		(*read Parametervalue*)
		3:	iReadValue	:=DWORD_TO_WORD(SHR(iParameterReadValue,((iSlaveaddress-(iParametergroup*2))-1)*16));
			IF (NOT bStart) OR ( bCycleMode) THEN
				fbParameterinterface(bStart			:=FALSE,
								stParameterBuffer	:=stParameterBuffer);
				IF (NOT fbParameterinterface.bBusy) THEN
					istate	:=10;
				END_IF
			ELSE
				istate	:=2;
			END_IF

			(*Quit*)
		10:	bBusy	:=FALSE;
			IF (NOT bStart) THEN
				istate	:=0;
			END_IF

	ELSE
		;
	END_CASE
END_FUNCTION_BLOCK

(* POU FB_ASI_Processdata_digital, ST *)
(*********************************************************************************************************

NAME..............	:	FB_Processdata_digital
DATE...............	:	21.03.2002
AUTHOR........	:	G.Sieder (Beckhoff Industrieelektronik)

DESCRIPTION:	FB for Read/Write digital data from/to one Slave

HISTORY:	
21.03.2002	gs	start coding

*********************************************************************************************************)
FUNCTION_BLOCK FB_ASI_Processdata_digital
VAR_INPUT
	iSlaveaddress		:BYTE;
	iSlavevalue			:BYTE;
	bParametermode		:BOOL;		(*0: Read, 1: Write *)
	bCycleMode			:BOOL;		(*0: Acyclic , 1:Cyclic (permanent Read/Write) *)
	bCommMode			:BOOL;		(*0: Parameterzugriff, 1: ADS*)
	bRegComm			:BOOL;		(*Registerkommunikation: 0: Parameterzugriff, 1: Registerkommunikation *)
	bmaskAccess		:BOOL;		(*0:usual access, 1:mask access*)
	bStart				:BOOL;
END_VAR
VAR_OUTPUT
	bBusy				:BOOL;
	bErr					:BOOL;
	iErrornumber			:DWORD;
	iReadValue			:BYTE;
	iParametergroup		:WORD;
END_VAR
VAR_IN_OUT
	stParameterBuffer		:ST_ParameterBuffer;
END_VAR
VAR
	fbParameterinterface	:FB_ASI_Parameterinterface;
	TrigStart				:R_TRIG;
	iParametermask		:WORD;
	bHiWord				:BOOL;
	iParametervalue		:DWORD;
	iParameterReadValue	:DWORD;
	istate				:INT;
END_VAR
	CASE istate OF

		0:	TrigStart(clk:=bStart);
			IF TrigStart.Q THEN
				bBusy		:=TRUE;
				bErr			:=FALSE;
				iErrornumber	:=0;
				istate		:=1;
			END_IF

		(*prepare Parametervalue*)
		1:	iParametervalue	:=0;
			iParametergroup	:=iSlaveaddress/8;
			(*iParametervalue	:=SHL((iParametervalue+iSlavevalue),(((iSlaveaddress-(iParametergroup*8))-1)*4));*)
			IF bmaskAccess THEN
				IF (iSlaveaddress- iParametergroup*8)> 4 THEN
					iParametermask	:=DWORD_TO_WORD(ROL(iParametervalue,16));
					bHiWord			:=TRUE;
				ELSE
					iParametermask	:=DWORD_TO_WORD(iParametervalue);
				END_IF
			END_IF
			istate	:=2;

		(*write Parametervalue*)
		2:	fbParameterinterface(iParameternumber	:=iSlaveaddress/8+16#80,
							iParametervalue		:=iParametervalue,
							stParameterBuffer		:=stParameterBuffer,
							bHiWord				:=bHiWord,
							bmaskAccess		:=bmaskAccess,
							iParametermask		:=iParametermask,
							bParametermode		:=bParametermode,
							bCycleMode			:=bCycleMode,
							bCommMode			:=bCommMode,
							bRegComm			:=bRegComm,
							bStart				:=TRUE);
			IF (NOT fbParameterinterface.bBusy) OR bCycleMode THEN
				IF fbParameterinterface.bErr THEN
					bErr			:=TRUE;
					iErrornumber	:=fbParameterinterface.iErrornumber;
					fbParameterinterface(bStart			:=FALSE,
									stParameterBuffer	:=stParameterBuffer);
					istate	:=10;
				ELSIF (NOT bParametermode) OR bCycleMode THEN
					iParameterReadValue	:=fbParameterinterface.iParameterReadvalue;
					istate	:=3;
				ELSE
					istate	:=3;
				END_IF
			END_IF

		(*read Parametervalue*)
		3:	iReadValue	:=(DWORD_TO_BYTE(SHR(iParameterReadValue,((iSlaveaddress-(iParametergroup*8))*4)))) AND 2#00001111;
			IF (NOT bStart) OR ( NOT bCycleMode) THEN
				fbParameterinterface(bStart			:=FALSE,
								stParameterBuffer	:=stParameterBuffer);
				IF (NOT fbParameterinterface.bBusy) THEN
					istate	:=10;
				END_IF
			ELSE
				istate	:=2;
			END_IF

			(*Quit*)
		10:	bBusy	:=FALSE;
			IF (NOT bStart) THEN
				istate	:=0;
			END_IF

	ELSE
		;
	END_CASE
END_FUNCTION_BLOCK

(* POU FB_ASI_Projecting, ST *)
(*********************************************************************************************************

NAME..............	:	FB_Projecting
DATE...............	:	21.03.2002
AUTHOR........	:	G.Sieder (Beckhoff Industrieelektronik)

DESCRIPTION:	FB to Read/Write Parameters for the slave-configuration 

HISTORY:	
21.03.2002	gs	start coding

*********************************************************************************************************)
FUNCTION_BLOCK FB_ASI_Projecting
VAR_INPUT
	iSlaveaddress		:BYTE;
	iParametervalue		:DWORD;
	bIOValue			:BOOL;	(*Read/Write IO-value of a slave*)
	bIDCode				:BOOL;	(*Read/Write	ID-code of a slave*)
	bReadWrite			:BOOL;	(*0: Read, 1: Write*)
	bReadLPS			:BOOL;	(*Read List of all projected Slaves*)
	bStart				:BOOL;
END_VAR
VAR_OUTPUT
	bBusy				:BOOL;
	bErr					:BOOL;
	iErrornumber			:DWORD;
	iParameterReadvalue	:BYTE;	(*IO-value or ID-code of a slave*)
	iLPS				:DWORD;
END_VAR
VAR_IN_OUT
	stParameterBuffer		:ST_ParameterBuffer;
END_VAR
VAR
	iProjectingStep	:INT;
	TrigStart			:R_TRIG;
	iAddressFactor	:BYTE;
	iParameternumber	:WORD;
	iReadValue		:DWORD;
	fbParameterinterface	:FB_ASI_Parameterinterface;
END_VAR
	CASE iProjectingStep OF

	(*Idle*)
	0:	TrigStart(clk:=bStart);
		IF TrigStart.Q THEN
			bBusy				:=TRUE;
			bErr					:=FALSE;
			iErrornumber			:=0;
			iProjectingStep		:=1;
		END_IF

	(*generate Parameternumber*)
	1:	iAddressFactor	:=iSlaveaddress / 8;
		IF bIOValue THEN
			iParameternumber	:=16#40+iAddressFactor;
		ELSIF bIDCode THEN
			iParameternumber	:=16#48+iAddressFactor;
		ELSIF bReadLPS	THEN
			iParameternumber	:=16#A8;
		END_IF
		iProjectingStep	:=2;

	(*write Parameter to ASI-Master*)
	2:	fbParameterinterface(iParameternumber	:=iParameternumber,
							iParametervalue	:=iParametervalue,
							stParameterBuffer	:=stParameterBuffer,
							bParametermode	:=bReadWrite,
							bCycleMode		:=TRUE,
							bStart			:=TRUE);
			IF (NOT fbParameterinterface.bBusy)  THEN
				IF fbParameterinterface.bErr THEN
					bErr			:=TRUE;
					iErrornumber	:=fbParameterinterface.iErrornumber;
					iProjectingStep	:=10;
				ELSE
					iReadValue	:=fbParameterinterface.iParameterReadvalue;
					iProjectingStep	:=3;
				END_IF
				fbParameterinterface(bStart			:=FALSE,
								stParameterBuffer	:=stParameterBuffer);
			END_IF

	(*generate ParameterReadvalue*)
	3:	IF bReadLPS THEN
			iParameterReadvalue	:=0;
			iLPS				:=iReadValue;
		ELSE
			iParameterReadvalue	:=DWORD_TO_BYTE(SHR(iReadValue,((iSlaveaddress-iAddressFactor*8)*4))) AND 2#00001111;
			iLPS	:=0;
		END_IF
		iProjectingStep	:=10;

	(*Quit*)
	10:	bBusy			:=FALSE;
		bStart			:=FALSE;
		iProjectingStep	:=0;

	ELSE
		;
	END_CASE
END_FUNCTION_BLOCK

(* POU FB_ASI_ReadParameter, ST *)
(*********************************************************************************************************

NAME..............	:	FB_ReadParameter
DATE...............	:	21.03.2002
AUTHOR........	:	G.Sieder (Beckhoff Industrieelektronik)

DESCRIPTION:	FB to read Parameters 

HISTORY:	
21.03.2002	gs	start coding

*********************************************************************************************************)
FUNCTION_BLOCK FB_ASI_ReadParameter
VAR_INPUT
	iParameternumber		:WORD;
	bCycleMode			:BOOL;		(*0: Acyclic , 1:Cyclic (permanent Read/Write) *)
	bStart				:BOOL;
END_VAR
VAR_OUTPUT
	bBusy				:BOOL;
	bErr					:BOOL;
	iErrornumber			:DWORD;
	iParameterReadvalue	:DWORD;
END_VAR
VAR_IN_OUT
	stParameterBuffer		:ST_ParameterBuffer;
END_VAR
VAR
	iReadStep	:INT;
	TrigStart		:R_TRIG;
	fbParameterinterface	:FB_ASI_Parameterinterface;
END_VAR
CASE iReadStep OF

	(*Idle*)
	0:	TrigStart(clk:=bStart);
		IF TrigStart.Q THEN
			bBusy				:=TRUE;
			bErr					:=FALSE;
			iErrornumber			:=0;
			iReadStep			:=1;
		END_IF

	(*wite Parameters to ASI-Master*)
	1:	fbParameterinterface(iParameternumber	:=iParameternumber,
							stParameterBuffer	:=stParameterBuffer,
							bParametermode	:=FALSE,
							bCycleMode		:=bCycleMode,
							bStart			:=TRUE);
		(*read Parameters *)
		IF (NOT fbParameterinterface.bBusy) OR  bCycleMode THEN
			IF fbParameterinterface.bErr THEN
				bErr			:=TRUE;
				iErrornumber	:=fbParameterinterface.iErrornumber;
				iReadStep	:=5;
			ELSE
				iParameterReadvalue	:=fbParameterinterface.iParameterReadvalue;
				IF (NOT bCycleMode) OR (NOT bStart) THEN
					iReadStep	:=5;
				ELSE
					iReadStep	:=1;
				END_IF
			END_IF
		END_IF

	5:	fbParameterinterface(bStart			:=FALSE,
						stParameterBuffer	:=stParameterBuffer);
		IF (NOT fbParameterinterface.bBusy) THEN
			iReadStep	:=10;
		END_IF

	(*Quit*)
	10:	bBusy			:=FALSE;
		bStart			:=FALSE;
		iReadStep	:=0;

	ELSE
		;
	END_CASE
END_FUNCTION_BLOCK

(* POU FB_ASI_SlaveDiag, ST *)
(*********************************************************************************************************

NAME..............	:	FB_WriteParameter
DATE...............	:	21.03.2002
AUTHOR........	:	G.Sieder (Beckhoff Industrieelektronik)

DESCRIPTION:	FB for cyclic slave-diagnosis

HISTORY:	
21.03.2002	gs	start coding
03.09.2002	gs	replace bStop by bCycleMode
*********************************************************************************************************)
FUNCTION_BLOCK FB_ASI_SlaveDiag
VAR_INPUT
	iSlaveaddress		:BYTE;
	iCounter				:INT;		(*1:PhysicalFaultCounter,  2:TimeoutCounter,  3:ResponseCounter,  4:Leave-DataExchCounter,  5:DataExch-FailedCounter *)
	bCounterReset		:BOOL;
	bReadLES			:BOOL;		(*Read List of all detected Slaves*)
	bReadLAS			:BOOL;		(*Read List of all activated Slaves*)
	bCycleMode			:BOOL;		(*0: Acyclic , 1:Cyclic (permanent Read/Write) *)
	bStart				:BOOL;

END_VAR
VAR_OUTPUT
	bBusy				:BOOL;
	bErr					:BOOL;
	iErrornumber			:DWORD;
	iCounterValue		:WORD;		(*Counter of a slave*)
	iSlaveList			:DWORD;	(*LES or LAS of all Slaves*)
END_VAR
VAR_IN_OUT
	stParameterBuffer		:ST_ParameterBuffer;
END_VAR
VAR
	iDiagStep			:INT;
	TrigStart				:R_TRIG;
	iAddressFactor		:BYTE;
	iParameternumber		:WORD;
	iReadValue			:DWORD;
	fbParameterinterface	:FB_ASI_Parameterinterface;

	TimerResetCounter	:TON;
END_VAR
	CASE iDiagStep OF

	(*Idle*)
	0:	TrigStart(clk:=bStart);
		IF TrigStart.Q THEN
			bBusy				:=TRUE;
			bErr					:=FALSE;
			iErrornumber			:=0;
			iDiagStep			:=1;
		END_IF

	(*generate Parameternumber*)
	1:	iAddressFactor	:=iSlaveaddress / 2;
		IF bReadLES	THEN
			iParameternumber	:=16#B0;
		ELSIF bReadLAS THEN
			iParameternumber	:=16#B8;
		ELSE
			CASE iCounter OF
				1:	iParameternumber	:=16#140+iAddressFactor;
				2:	iParameternumber	:=16#160+iAddressFactor;
				3:	iParameternumber	:=16#180+iAddressFactor;
				4:	iParameternumber	:=16#1A0+iAddressFactor;
				5:	iParameternumber	:=16#1C0+iAddressFactor;
			ELSE
				;
			END_CASE
		END_IF
		iDiagStep	:=2;

	(*write Parameter to ASI-Master*)
	2:	fbParameterinterface(iParameternumber		:=iParameternumber,
							stParameterBuffer		:=stParameterBuffer,
							iParametervalue		:=0,
							bParametermode		:=bCounterReset,
							bCycleMode			:=TRUE,
							bStart				:=TRUE);
				IF fbParameterinterface.bErr THEN
					bErr			:=TRUE;
					iErrornumber	:=fbParameterinterface.iErrornumber;
					iDiagStep	:=10;
				ELSE
					iReadValue	:=fbParameterinterface.iParameterReadvalue;
					iDiagStep	:=3;
				END_IF
				TimerResetCounter(in:=bCounterReset,pt:=t#200ms);
				IF TimerResetCounter.Q THEN
					bCounterReset		:=FALSE;
					TimerResetCounter.IN 	:=FALSE;
				END_IF

	(*generate ParameterReadvalue*)
	3:	fbParameterinterface(stParameterBuffer	:=stParameterBuffer);
		IF bReadLES OR bReadLAS THEN
			iCounterValue	:=0;
			iSlaveList		:=iReadValue;
		ELSE
			iCounterValue	:=DWORD_TO_WORD(SHR(iReadValue,((iSlaveaddress-iAddressFactor*2)*16)));
			iSlaveList	:=0;
		END_IF
		IF (NOT bStart) THEN
			fbParameterinterface(bStart	:=FALSE,
							stParameterBuffer	:=stParameterBuffer);
			IF (NOT fbParameterinterface.bBusy) THEN
				iDiagStep	:=10;
			END_IF
		ELSE
			iDiagStep	:=2;
		END_IF

	(*Quit*)
	10:	bBusy		:=FALSE;
		bStart		:=FALSE;
		iDiagStep	:=0;

	ELSE
		;
	END_CASE
END_FUNCTION_BLOCK

(* POU FB_ASI_WriteParameter, ST *)
(*********************************************************************************************************

NAME..............	:	FB_WriteParameter
DATE...............	:	21.03.2002
AUTHOR........	:	G.Sieder (Beckhoff Industrieelektronik)

DESCRIPTION:	FB to write Parameters 

HISTORY:	
21.03.2002	gs	start coding
03.09.2002	gs	Output ReadValue removed
*********************************************************************************************************)
FUNCTION_BLOCK FB_ASI_WriteParameter
VAR_INPUT
	iParameternumber		:WORD;
	iParametervalue		:DWORD;
	bStart				:BOOL;
END_VAR
VAR_OUTPUT
	bBusy				:BOOL;
	bErr					:BOOL;
	iErrornumber			:DWORD;
END_VAR
VAR_IN_OUT
	stParameterBuffer		:ST_ParameterBuffer;
END_VAR
VAR
	iWriteStep	:INT;
	TrigStart		:R_TRIG;
	fbParameterinterface	:FB_ASI_Parameterinterface;
END_VAR
	CASE iWriteStep OF

	(*Idle*)
	0:	TrigStart(clk:=bStart);
		IF TrigStart.Q THEN
			bBusy				:=TRUE;
			bErr					:=FALSE;
			iErrornumber			:=0;
			iWriteStep			:=1;
		END_IF

	(*wite Parameters to ASI-Master*)
	1:	fbParameterinterface(iParameternumber	:=iParameternumber,
							iParametervalue	:=iParametervalue,
							stParameterBuffer	:=stParameterBuffer,
							bParametermode	:=TRUE,
							bCycleMode		:= FALSE,
							bStart			:=TRUE);
		IF  fbParameterinterface.bBusy  THEN
			iWriteStep	:=5;
		END_IF


	5:	fbParameterinterface(stParameterBuffer	:=stParameterBuffer);
		IF (NOT fbParameterinterface.bBusy) THEN
			IF fbParameterinterface.bErr THEN
				bErr			:=TRUE;
				iErrornumber	:=fbParameterinterface.iErrornumber;
			END_IF
			iWriteStep	:=10;
		END_IF

	(*Quit*)
	10:	bBusy			:=FALSE;
		bStart			:=FALSE;
		iWriteStep	:=0;

	ELSE
		;
	END_CASE
END_FUNCTION_BLOCK

(* POU FB_ASI_WriteReadParameter, ST *)
(*********************************************************************************************************

NAME..............	:	FB_WriteReadParameter
DATE...............	:	18.08.2003
AUTHOR........	:	G.Sieder (Beckhoff Industrieelektronik)

DESCRIPTION:	FB to write Parameters with answer 

HISTORY:	
18.08.2003	gs	start coding

*********************************************************************************************************)
FUNCTION_BLOCK FB_ASI_WriteReadParameter
VAR_INPUT
	iParameternumber		:WORD;
	iParametervalue		:DWORD;
	bStart				:BOOL;
END_VAR
VAR_OUTPUT
	bBusy				:BOOL;
	bErr					:BOOL;
	iParameterReadValue	:DWORD;
	iErrornumber			:DWORD;
END_VAR
VAR_IN_OUT
	stParameterBuffer		:ST_ParameterBuffer;
END_VAR
VAR
	iWriteStep	:INT;
	TrigStart		:R_TRIG;
	fbParameterinterface	:FB_ASI_Parameterinterface;
END_VAR
	CASE iWriteStep OF

	(*Idle*)
	0:	TrigStart(clk:=bStart);
		IF TrigStart.Q THEN
			bBusy				:=TRUE;
			bErr					:=FALSE;
			iErrornumber			:=0;
			iWriteStep			:=1;
		END_IF

	(*wite Parameters to ASI-Master*)
	1:	fbParameterinterface(iParameternumber	:=iParameternumber,
							iParametervalue	:=iParametervalue,
							stParameterBuffer	:=stParameterBuffer,
							bParametermode	:=TRUE,
							bCycleMode		:= FALSE,
							bStart			:=TRUE);
		IF  fbParameterinterface.bBusy  THEN
			iWriteStep	:=5;
		END_IF


	5:	fbParameterinterface(stParameterBuffer	:=stParameterBuffer);
		IF (NOT fbParameterinterface.bBusy) THEN
			IF fbParameterinterface.bErr THEN
				bErr			:=TRUE;
				iErrornumber	:=fbParameterinterface.iErrornumber;
				iParameterReadValue	:=0;
			ELSE
				iParameterReadValue	:=fbParameterinterface.iParameterReadvalue;
			END_IF
			iWriteStep	:=10;
		END_IF

	(*Quit*)
	10:	bBusy			:=FALSE;
		bStart			:=FALSE;
		iWriteStep	:=0;

	ELSE
		;
	END_CASE
END_FUNCTION_BLOCK

(* POU FB_AX2000_AXACT, ST *)
FUNCTION_BLOCK FB_AX2000_AXACT
VAR_INPUT
	bMode_DigitalSpeed	: BOOL;			(*OP-Mode digital speed instead of Positioning*)
	iDigitalSpeed			: DWORD;			(*digital speed if OP-Mode = digital speed*)
	iVelocity				: DWORD;		(*Velocity*)
	iPosition				: DINT;			(*Position*)
	imotion_tasknumber	: WORD;			(*number of EEPROM-saved motion-task*)
	imotion_blocktype		: WORD;			(*optional Parameters of motion tasks*)
	bStart				: BOOL;			(*START*)
	bStop				: BOOL;			(*STOP*)
	bShortStop			: BOOL;			(*1: break of motion task, 0: continue same motion task*)
	bErrorResume		: BOOL;			(*Error resume*)
	tTimeOut				: TIME:=t#5s;
END_VAR
VAR_OUTPUT

	bBusy				: BOOL;
	bError				: BOOL;			(*Errorstatus of Servo*)
	bTimeOutErr			: BOOL;

END_VAR
VAR
	i16State:				INT;
	icheckStatus:			WORD;
	icheckControlWord:	WORD;			(*ControlWord for Servo*)

	bServoReady:		BOOL;			(*readyFlag for HSW*)
	TrigStart:				R_TRIG;
	TrigTimeOut:			R_TRIG;
	bResetServo:			BOOL;			(*first move of Servo after Start/Restart*)

	TimerTimeOut		:TON;
	bTimeOutStart		:BOOL;

	iHighByte			:BYTE;
	iLowByte				:BYTE;
	icheckByteSwaping	:WORD;
	bMapInOutputs		:BOOL;
	bShortStop_check		:BOOL;

	(*virtual Input/Output*)
	stPZD_IN:		ST_PZD_IN;
	stPZD_OUT:		ST_PZD_OUT;
END_VAR
VAR_IN_OUT
	stPZDIN:		ST_PZD_IN;			(*Data from NC*)
	stPZDOUT:		ST_PZD_OUT;			(*Data to NC*)
END_VAR
	a_MapInputs();			(*mapping of real Inputs to virtual Inputs by swaping LowByte and HighByte*)
	a_RW_CtrlWord();			(*AXACT-controls*)
	a_MapOutputs();			(*mapping of virtual Outputs to real Outputs by swaping LowByte and HighByte*)
END_FUNCTION_BLOCK
ACTION a_MapInputs:
stPZD_IN.wSTW		:=ROL(stPZDIN.wSTW,8);
stPZD_IN.wHIW		:=ROL(stPZDIN.wHIW,8);
stPZD_IN.PZD3		:=ROL(stPZDIN.PZD3,8);
stPZD_IN.PZD4		:=ROL(stPZDIN.PZD4,8);
stPZD_IN.PZD5		:=ROL(stPZDIN.PZD5,8);
stPZD_IN.PZD6		:=ROL(stPZDIN.PZD6,8);
END_ACTION
ACTION a_MapOutputs:
IF bMapInOutputs THEN
	stPZDOUT.wCtrlW		:=ROL(stPZD_OUT.wCtrlW,8);
	stPZDOUT.PZD2		:=ROL(stPZD_OUT.PZD2,8);
	stPZDOUT.PZD3		:=ROL(stPZD_OUT.PZD3,8);
	stPZDOUT.PZD4		:=ROL(stPZD_OUT.PZD4,8);
	stPZDOUT.PZD5		:=ROL(stPZD_OUT.PZD5,8);
	stPZDOUT.PZD6		:=ROL(stPZD_OUT.PZD6,8);
END_IF
END_ACTION
ACTION a_RW_CtrlWord:
	bMapInOutputs	:= TRUE;

	(* Errorstatus*)
	icheckStatus:=2#00000000_00001000;
	IF (stPZD_IN.wSTW AND icheckStatus)<>0 THEN
		i16State:=10;
	END_IF

	(*short break of a motion task*)
	IF bShortStop AND (NOT bShortStop_check)THEN
		stPZD_OUT.wCtrlW:=stPZD_OUT.wCtrlW AND 2#1111111111011111;
		bShortStop_check	:=TRUE;
	ELSIF (NOT bShortStop) AND bShortStop_check THEN
		bShortStop_check	:=FALSE;
		IF (NOT bStart) THEN
			i16State			:= 11;
			bBusy			:= FALSE;
		ELSE
			stPZD_OUT.wCtrlW:=stPZD_OUT.wCtrlW OR 2#0000000000100000;
		END_IF
	END_IF

	(*Stophandling*)
	IF  bStop THEN
		stPZD_OUT.wCtrlW:=2#0000000000000101;
		bBusy			:= FALSE;
		bStart			:= FALSE;
		bMapInOutputs	:= TRUE;
		i16State			:= 11;
	END_IF

	(*TimeOut*)
	IF (NOT bMode_DigitalSpeed) THEN
		TrigTimeOut(clk:=bStart);
		IF TrigTimeOut.Q THEN
			bTimeOutStart	:=TRUE;
			bTimeOutErr		:= FALSE;
			bError			:= FALSE;
		END_IF
		IF bBusy THEN
			TimerTimeOut(IN:= FALSE, PT:= tTimeOut );
			bTimeOutStart	:=FALSE;
		ELSE
			TimerTimeOut(IN:= bTimeOutStart, PT:= tTimeOut );
		END_IF
		IF TimerTimeOut.Q THEN
			bTimeOutErr		:=TRUE;
			bTimeOutStart	:= FALSE;
			bServoReady	:= FALSE;
			i16State			:= 11;
		END_IF
	END_IF

	CASE i16State OF

		(*Initialisierung*)
	0:	bServoReady:= 	FALSE;
		bResetServo:=	TRUE;
		i16State:= i16State+1;

		(*Einschaltsperre*)
	1:	stPZD_OUT.wCtrlW:=2#0000000000000000;
		icheckStatus:=2#0000000001000000;
		IF (stPZD_IN.wSTW AND icheckStatus)<>0 THEN
			stPZD_OUT.wCtrlW:=2#0000000000000110;
			bServoReady:= FALSE;
			i16State:= i16State+1;
		END_IF

		(*einschaltbereit*)
	2:	icheckStatus:=2#0000001000000001;
		IF (stPZD_IN.wSTW AND icheckStatus)<>0 THEN
			stPZD_OUT.wCtrlW:=2#0000000000000111;
			bServoReady:= FALSE;
			i16State:= i16State+1;
		END_IF

		(*betriebsbereit*)
	3:	icheckStatus:=2#0000001000100011;
		IF (stPZD_IN.wSTW AND icheckStatus)<>0 THEN
			stPZD_OUT.wCtrlW:=2#0000010000111111;
			i16State:= i16State+1;
		END_IF

		(*Betrieb freigegeben*)
	4:	icheckStatus:=2#0000001000100111;
		IF (stPZD_IN.wSTW AND icheckStatus)<>0 THEN
			i16State:= i16State+1;
		END_IF

		(*benutzerdefinierte Daten übertragen*)
	5:	TrigStart(clk:=bStart);
		bMapInOutputs	:= FALSE;
		IF TrigStart.Q THEN
			bMapInOutputs:= TRUE;
			a_RW_PZD();
			bError		:= FALSE;
			bTimeOutErr	:= FALSE;
			bResetServo	:= FALSE;
		END_IF
		IF (NOT bResetServo) THEN
			icheckStatus:=2#0010000000000000;
			IF (stPZD_IN.wSTW AND icheckStatus)<>0 THEN
				;
			ELSE
				bBusy	:= TRUE;
				i16State:= 6;
			END_IF
		END_IF

	6:	icheckStatus:=2#0010000000000000;
		IF (stPZD_IN.wSTW AND icheckStatus)<>0 THEN
			bBusy	:= FALSE;
			i16State:= 5;
		END_IF
		IF bMode_DigitalSpeed THEN
			stPZD_OUT.PZD3	:=DWORD_TO_WORD(iDigitalSpeed*140);
			stPZD_OUT.PZD2	:=DWORD_TO_WORD(SHR((iDigitalSpeed*140),16));
		END_IF

		(* Errorhandling*)
	10:	bError			:= TRUE;
		bBusy			:= FALSE;
		bServoReady	:= FALSE;
		IF BErrorResume THEN
			stPZD_OUT.wCtrlW:=2#0000010010001111;
			i16State:=11;
		END_IF

	11:	IF (NOT bStart) THEN
			i16State:=0;
		END_IF

END_CASE
END_ACTION
ACTION a_RW_PZD:
IF bMode_DigitalSpeed THEN
	stPZD_OUT.PZD3	:=DWORD_TO_WORD(iDigitalSpeed*140);
	stPZD_OUT.PZD2	:=DWORD_TO_WORD(SHR((iDigitalSpeed*140),16));
	icheckControlWord:=2#0000000001000000;
	IF (icheckControlWord AND stPZD_OUT.wCtrlW)<>0 THEN
		stPZD_OUT.wCtrlW:=16#443F;
	ELSE
		stPZD_OUT.wCtrlW:=16#447F;
	END_IF
ELSIF (imotion_tasknumber <> 0) THEN
	stPZD_OUT.PZD2	:=imotion_tasknumber;
	icheckControlWord:=2#0000000001000000;
	IF (icheckControlWord AND stPZD_OUT.wCtrlW)<>0 THEN
		stPZD_OUT.wCtrlW:=16#043F;
	ELSE
		stPZD_OUT.wCtrlW:=16#047F;
	END_IF
ELSIF (iVelocity<>0) THEN
	stPZD_OUT.PZD3	:=DWORD_TO_WORD(iVelocity);
	stPZD_OUT.PZD2	:=DWORD_TO_WORD(SHR(iVelocity,16));
	stPZD_OUT.PZD5	:=DWORD_TO_WORD(DINT_TO_DWORD( iPosition ));
	stPZD_OUT.PZD4	:=DWORD_TO_WORD(SHR(DINT_TO_DWORD( iPosition ),16));
	stPZD_OUT.PZD6	:=imotion_blocktype;
	icheckControlWord:=2#0000000001000000;
	IF (icheckControlWord AND stPZD_OUT.wCtrlW)<>0 THEN
		stPZD_OUT.wCtrlW:=16#443F;
	ELSE
		stPZD_OUT.wCtrlW:=16#447F;
	END_IF
END_IF
END_ACTION

(* POU FB_AX2000_JogMode, ST *)
FUNCTION_BLOCK FB_AX2000_JogMode
VAR_INPUT
	bStart		: BOOL;
	bStop		: BOOL;
	iBasicVelo	: INT;				(*BasicVelocity*)
	tTimeOut		: TIME:=t#5s;

END_VAR
VAR_OUTPUT
	bBusy		: BOOL;
	bErr			: BOOL;
	bTimeOutErr	: BOOL;

END_VAR
VAR_IN_OUT
	stPZDIN			: ST_PZD_IN;			(*Data from NC*)
	stPZDOUT		: ST_PZD_OUT;		(*Data to NC*)
END_VAR
VAR
	i16state			: INT;

	icheckStatus		: DWORD;
	TrigTimeOut		: R_TRIG;
	bTimeOutStart	: BOOL;
	TimerTimeOut	: TON;
	bMapInOutputs	: BOOL;
	(*virtual Input/Output*)
	stPZD_IN:		ST_PZD_IN;
	stPZD_OUT:		ST_PZD_OUT;

END_VAR
	a_MapInputs();

	(* Errorstatus*)
	icheckStatus:=2#00000000_00001000;
	IF (stPZD_IN.wSTW AND icheckStatus)<>0 THEN
		bErr	:= TRUE;
		i16State:=10;
	END_IF

	(*TimeOut*)
	TrigTimeOut(clk:=bStart);
	IF TrigTimeOut.Q THEN
		bTimeOutStart	:=TRUE;
	END_IF
	IF bBusy THEN
		TimerTimeOut(IN:= FALSE, PT:= tTimeOut );
		bTimeOutStart	:=FALSE;
	ELSE
		TimerTimeOut(IN:= bTimeOutStart, PT:= tTimeOut );
	END_IF
	IF TimerTimeOut.Q THEN
		TimerTimeOut(IN:= FALSE, PT:= tTimeOut );
		bTimeOutErr		:=TRUE;
		bTimeOutStart	:= FALSE;
		i16State			:= 10;
	END_IF

	CASE i16state OF

	0:	IF bStart THEN
			bErr				:= FALSE;
			bTimeOutErr		:= FALSE;
			i16state			:= 1;
		END_IF

	1:	stPZD_OUT.PZD2	:=iBasicVelo;
		stPZD_OUT.wCtrlW:=(ROL(stPZDOUT.wCtrlW,8))+16#100;
		bMapInOutputs	:= TRUE;
		i16state	:= 2;

	2:	icheckStatus:=2#00100010_00000000;
		IF (stPZD_IN.wSTW AND icheckStatus)=0 OR  (stPZD_IN.wSTW AND icheckStatus)=16#2200 THEN
			;
		ELSE
			bBusy	:=TRUE;
			i16state	:= 3;
		END_IF

	3:	IF bStop THEN
			stPZD_OUT.wCtrlW:=(ROL(stPZDOUT.wCtrlW,8))-16#100;
			i16state	:= 10;
		END_IF

	10:	bBusy			:=FALSE;
		bMapInOutputs	:=FALSE;
		IF (NOT bstart) THEN
			i16state	:= 0;
		END_IF

	END_CASE

	a_MapOutputs();
END_FUNCTION_BLOCK
ACTION a_MapInputs:
	stPZD_IN.wSTW		:=ROL(stPZDIN.wSTW,8);
	stPZD_IN.wHIW		:=ROL(stPZDIN.wHIW,8);
	stPZD_IN.PZD3		:=ROL(stPZDIN.PZD3,8);
	stPZD_IN.PZD4		:=ROL(stPZDIN.PZD4,8);
	stPZD_IN.PZD5		:=ROL(stPZDIN.PZD5,8);
	stPZD_IN.PZD6		:=ROL(stPZDIN.PZD6,8);
END_ACTION
ACTION a_MapOutputs:
IF bMapInOutputs THEN
	stPZDOUT.wCtrlW		:=ROL(stPZD_OUT.wCtrlW,8);
	stPZDOUT.PZD2		:=ROL(stPZD_OUT.PZD2,8);
	stPZDOUT.PZD3		:=ROL(stPZD_OUT.PZD3,8);
	stPZDOUT.PZD4		:=ROL(stPZD_OUT.PZD4,8);
	stPZDOUT.PZD5		:=ROL(stPZD_OUT.PZD5,8);
	stPZDOUT.PZD6		:=ROL(stPZD_OUT.PZD6,8);
END_IF
END_ACTION

(* POU FB_AX2000_Parameter, ST *)
FUNCTION_BLOCK FB_AX2000_Parameter
VAR_INPUT
	iSlaveAddress:	BYTE := 0;			(* Station Address of the Slave *)
	iPnu:				WORD := 16#03A2;	(* Parameter-Number *)
	nAxis:				BYTE := 1;			(* Number of Axis *)
	iLength:			BYTE := 4;			(* Length of the parameter (2 or 4) *)
	iSubindex:			BYTE := 1;			(*Subindex*)
	iParameterValue:	DWORD := 2;			(* Parameter value *)
	iFC310xDeviceId: 	WORD := 1;			(* Device-ID of the FCxxxx *)
	bStartRead:		BOOL;				(* StartFlag to start the PKW-Read *)
	bStartWrite:		BOOL;				(* StartFlag to start the PKW-Write *)
	tTimeOut:			TIME := DEFAULT_ADS_TIMEOUT;
END_VAR
VAR_OUTPUT
	bBusy				:BOOL;
	iErrorId			:DWORD;
	iReadValue		:DINT;
END_VAR
VAR
	iError:					DWORD;
	fbReadPkw:				FB_FCxxxxDpv0PkwRead;
	fbWritePkw: 				FB_FCxxxxDpv0PkwWrite;

END_VAR
IF bStartRead OR bStartWrite THEN
	IF iLength<>2 THEN
		iLength:= 4;
	END_IF
	
	(* PKW-Read with DPV0  for Stoever-Drive (ArrayCodesNotSupported and Subindex in Octet 3 must be set) *)
	fbReadPkw(bStartFlag := bStartRead, iStationAdd := iSlaveAddress, iDeviceId := iFC310xDeviceId,nAxis := nAxis, iPnu := iPnu, iSubindex := iSubindex, iLength := iLength, bArrayCodesNotSupported := TRUE, bSubindexInOctet3 := TRUE, tTimeOut:=tTimeOut);
	IF (bStartRead AND NOT fbReadPkw.bBusy) THEN
		iError := fbReadPkw.iErrorId;
		iReadValue := fbReadPkw.iReadValue;
		bStartRead := FALSE;
	END_IF;
	
	(* PKW-Write with DPV0  for Stoever-Drive (ArrayCodesNotSupported and Subindex in Octet 3 must be set) *)
	fbWritePkw(bStartFlag := bStartWrite, iStationAdd := iSlaveAddress, iDeviceId := iFC310xDeviceId, nAxis := nAxis, iPnu := iPnu, iSubindex := iSubindex, iLength := iLength, iWriteValue := iParameterValue, bArrayCodesNotSupported := TRUE, bSubindexInOctet3 := TRUE, tTimeOut:=tTimeOut);
	IF (bStartWrite AND NOT fbWritePkw.bBusy) THEN
		iError := fbWritePkw.iErrorId;
		bStartWrite := FALSE;
	END_IF;

	bBusy:=fbReadPkw.bBusy OR fbWritePkw.bBusy;
	iErrorId:=iError;
	(*iReadValue:=iParameterValue;*)
END_IF
END_FUNCTION_BLOCK

(* POU FB_FCxxxxDpv0PkwRead, ST *)
FUNCTION_BLOCK FB_FCxxxxDpv0PkwRead
VAR_INPUT
	bStartFlag:BOOL;					(* StartFlag to start the PKW-Read *)
	iStationAdd: BYTE;				(* Station Address of the Slave *)
	iDeviceId: WORD;					(* Device-ID of the FCxxxx *)
	nAxis: BYTE;						(* Number of Axis *)
	iPnu: WORD;						(* Parameter-Number *)
	iSubindex: BYTE;					(* Subindex  *)
	iLength:BYTE;					(* Length of the parameter (2 or 4) *)
	bArrayCodesNotSupported: BOOL;	(* if the drive does not support the ARRAY-AKs 6,7 and 8, this flag should be set (then the AKs 1,2,3 will be used for Arrays) *)
	bSubindexInOctet3:BOOL;			(* if the drive needs the subindex in Octet 3 (ProfiDrive 2.0), this flag should be set *)
	tTimeOut		: TIME;
END_VAR
VAR_OUTPUT
	bBusy:BOOL;			(* Reading is busy *)
	iErrorId:DWORD;
	iReadValue:DWORD;	(* Parameter value *)
END_VAR
VAR
	fbRead:ADSREAD;
	fbDevNetId:IOF_GetDeviceNetId;
	istate:WORD := 0;
	sDevNetId:STRING(23);
	iIdxGrp: DWORD;
	iport:WORD;
	iParameterValue:DWORD;
END_VAR
CASE istate OF

	0:	(*Idle*)
		IF bStartFlag THEN
			bBusy	:=TRUE;
			istate := 1;
		END_IF

	1:	(* Get Net-ID of FCxxxx-Device *)
		fbDevNetId(NETID := '', DEVICEID := iDeviceId, START := TRUE,  TMOUT := T#1s);
		IF (NOT fbDevNetId.BUSY) THEN
			IF (NOT fbDevNetId.Err) THEN
				sDevNetId := fbDevNetId.DeviceNetId;
				istate := 2;
			ELSE
				iErrorId		:=fbDevNetId.ERRID;
				bStartFlag	:=FALSE;
				bBusy		:=FALSE;
				istate := 0;
			END_IF
			fbDevNetId(NETID := '', DEVICEID := iDeviceId, START := FALSE,  TMOUT := T#1s);
		END_IF

	2:	(* Read Parameter if StartFlag is set *)
		iport := iStationAdd;
		iport := iport + 16#1000;
		iIdxGrp := nAxis;
		iIdxGrp := SHL(iIdxGrp, 28);
		iIdxGrp := iIdxGrp +iPnu;
		IF (bArrayCodesNotSupported) THEN
			iIdxGrp := iIdxGrp + 16#8000000;
		END_IF
		IF (bSubindexInOctet3) THEN
			iIdxGrp := iIdxGrp + 16#4000000;
		END_IF
		fbRead(	NETID := sDevNetId, PORT := iport, IDXGRP := iIdxGrp, IDXOFFS := iSubindex, LEN := iLength,
				DESTADDR := ADR(iParameterValue), READ := bStartFlag, TMOUT := tTimeOut);
		istate := 3;

	3:	fbRead(	NETID := sDevNetId, PORT := iport, IDXGRP := iIdxGrp, IDXOFFS := iSubindex, LEN := iLength,
				DESTADDR := ADR(iParameterValue), READ := bStartFlag, TMOUT := tTimeOut);
		IF (NOT FbRead.BUSY) OR fbRead.Err THEN
			iErrorId := FbRead.ERRID;
			iReadValue := iParameterValue;
			istate := 4;
		END_IF

	4:	(* There must be a rising edge on the READ-input of ADSREAD to start the next reading *)
		fbRead(	NETID := sDevNetId, PORT := iport, IDXGRP := iIdxGrp, IDXOFFS := iSubindex, LEN := iLength,
				DESTADDR := ADR(iParameterValue), READ := FALSE, TMOUT := tTimeOut);
		bBusy 		:= FALSE;
		bStartFlag	:= FALSE;
		istate := 0;
END_CASE
END_FUNCTION_BLOCK

(* POU IOF_GetDeviceNetId, ST *)
FUNCTION_BLOCK IOF_GetDeviceNetId
VAR_INPUT
	NETID		: T_AmsNetId;
	DEVICEID	: UDINT;
	START		: BOOL;
	TMOUT		: TIME := DEFAULT_ADS_TIMEOUT;
END_VAR
VAR_OUTPUT
	BUSY		: BOOL;
	ERR			: BOOL;
	ERRID		: UDINT;
	DeviceNetId	: T_AmsNetId;
END_VAR
{library private}
VAR
	ADSREADEX1	: ADSREADEX := ( PORT:= AMSPORT_R0_IO, IDXOFFS:= 16#00000005 );
	RisingEdge	: R_TRIG;
	state		: BYTE;
	tmpNetId	: ARRAY[0..5] OF BYTE;
END_VAR
RisingEdge( CLK:=START );
IF RisingEdge.Q THEN
	state := 1;
END_IF
CASE state OF
	0:;(* idle state *)
	1:
		BUSY := TRUE;
		ERR := FALSE;
		ERRID := 0;
		DeviceNetId := '';
		MEMSET( ADR( tmpNetId ), 0, SIZEOF( tmpNetId ) );
		IF ( DEVICEID > 0 ) THEN
			ADSREADEX1( READ:=FALSE );
			ADSREADEX1( NETID:=NETID, IDXGRP:= 16#00005000 + DEVICEID,
						LEN:= SIZEOF( tmpNetId ), DESTADDR:= ADR( tmpNetId ),
						READ:=TRUE, TMOUT:= TMOUT );
			state := 2;
		ELSE
			ERR := TRUE;
			ERRID :=16#706;	(* Parameter value not correct! *)
			state := 100;
		END_IF
	2:
		ADSREADEX1( READ:=FALSE, BUSY=>BUSY, ERR=>ERR, ERRID=>ERRID );
		IF NOT BUSY THEN
			IF NOT ERR THEN
				IF ( ADSREADEX1.COUNT_R = SIZEOF( tmpNetId ) ) THEN (* check the read data length *)
					DeviceNetId := F_CreateAmsNetId( tmpNetid );
				ELSE
					ERR := TRUE;
					ERRID := 16#70B; (* 1803 invalid parameter value(s) *)
				END_IF
			END_IF
			state := 0;
		END_IF
	100:(* error state *)
		BUSY := FALSE;
		state := 0;
END_CASE
END_FUNCTION_BLOCK

(* POU FB_FCxxxxDpv0PkwWrite, ST *)
FUNCTION_BLOCK FB_FCxxxxDpv0PkwWrite
VAR_INPUT
	bStartFlag:BOOL;		(* StartFlag to start the PKW-REad *)
	iStationAdd: BYTE;		(* Station Address of the Slave *)
	iDeviceId: WORD;		(* Device-ID of the FCxxxx *)
	nAxis: BYTE;			(* Number of Axis *)
	iPnu: WORD;			(* Parameter-Number *)
	iSubindex: BYTE;		(* Subindex  *)
	iLength:BYTE;			(* Length of the parameter (2 or 4) *)
	iWriteValue:DWORD;	(* Parameter value *)
	bArrayCodesNotSupported: BOOL;	(* if the drive does not support the ARRAY-AKs 6,7 and 8, this flag should be set (then the AKs 1,2,3 will be used for Arrays) *)
	bSubindexInOctet3:BOOL;				(* if the drive needs the subindex in Octet 3 (ProfiDrive 2.0), this flag should be set *)
	tTimeOut		: TIME:=T#10s;
END_VAR
VAR_OUTPUT
	bBusy:BOOL;			(* Writing is busy *)
	iErrorId:DWORD;
END_VAR
VAR
	fbWrite:ADSWRITE;
	fbDevNetId:IOF_GetDeviceNetId;
	istate:WORD := 0;
	sDevNetId:STRING(23);
	iIdxGrp: DWORD;
	iport:WORD;
	iParameterValue:DWORD;
END_VAR
CASE istate OF

	0:	(*Idle*)
		IF bStartFlag THEN
			bBusy	:=TRUE;
			istate := 1;
		END_IF

	1:	(* Get Net-ID of FCxxxx-Device *)
		fbDevNetId(NETID := '', DEVICEID :=iDeviceId, START := TRUE,  TMOUT := T#1s);
		istate := 2;

	2:	fbDevNetId();
		IF (NOT fbDevNetId.BUSY) THEN
			IF (NOT fbDevNetId.Err) THEN
				sDevNetId := fbDevNetId.DeviceNetId;
				istate := 3;
			ELSE
				iErrorId		:=fbDevNetId.ERRID;
				bBusy		:=FALSE;
				bStartFlag	:=FALSE;
				istate := 0;
			END_IF
			fbDevNetId(NETID := '', DEVICEID := iDeviceId, START := FALSE,  TMOUT := T#1s);
		END_IF

	3:	(* Read Parameter if StartFlag is set *)
		iport := iStationAdd;
		iport := iport + 16#1000;
		iIdxGrp :=nAxis;
		iIdxGrp := SHL(iIdxGrp, 28);
		iIdxGrp := iIdxGrp + iPnu;
		IF (bArrayCodesNotSupported) THEN
			iIdxGrp := iIdxGrp + 16#8000000;
		END_IF
		IF (bSubindexInOctet3) THEN
			iIdxGrp := iIdxGrp + 16#4000000;
		END_IF
		iParameterValue :=iWriteValue;
		fbWrite(	NETID := sDevNetId, PORT := iport, IDXGRP := iIdxGrp, IDXOFFS := iSubindex, LEN := iLength,
				SRCADDR := ADR(iParameterValue), WRITE := bStartFlag, TMOUT := tTimeOut);
		istate := 4;

	4:	fbWrite();
		IF (NOT fbWrite.BUSY) OR fbWrite.Err THEN
			iErrorId := fbWrite.ERRID;
			istate := 5;
		END_IF

	5:	(* There must be a rising edge on the READ-input of ADSREAD to start the next reading *)
		fbWrite(	NETID := sDevNetId, PORT := iport, IDXGRP := iIdxGrp, IDXOFFS := iSubindex, LEN := iLength,
				SRCADDR := ADR(iParameterValue), WRITE := FALSE, TMOUT := tTimeOut);
		bBusy 		:= FALSE;
		bStartFlag	:= FALSE;
		istate := 0;
END_CASE
END_FUNCTION_BLOCK

(* POU FB_AX2000_Reference, ST *)
FUNCTION_BLOCK FB_AX2000_Reference
VAR_INPUT
	bSetRefPoint	: BOOL;		(* set Reference Point*)
	bCalibrStart	: BOOL;		(* start home running*)
	bCalibrStop	: BOOL;		(* stop home running*)
	iCalVelo		: WORD;		(* basic velocity of Calibration*)

END_VAR
VAR_OUTPUT
	bBusy	: BOOL;
	bErr	: BOOL;

END_VAR
VAR_IN_OUT
	stPZDIN		: ST_PZD_IN;	(*Data from NC*)
	stPZDOUT		: ST_PZD_OUT;(*Data to NC*)
END_VAR
VAR
	icheckStatus		: WORD;
	i16State			: INT;
	bMapInOutputs	: BOOL;
	(*virtual Input/Output*)
	stPZD_IN		: ST_PZD_IN;	(*Data from NC*)
	stPZD_OUT		: ST_PZD_OUT;(*Data to NC*)
END_VAR
	a_MapInputs();

	(* Errorstatus*)
	icheckStatus:=2#00000000_00001000;
	IF (stPZD_IN.wSTW AND icheckStatus)<>0 THEN
		i16State	:=9;
	END_IF

	CASE i16State OF

	(*start FB*)
	0:	IF bSetRefPoint OR bCalibrStart THEN
			bBusy			:= TRUE;
			bErr				:= FALSE;
			IF bSetRefPoint THEN
				i16State	:= 1;
			ELSE
				i16State	:= 3;
			END_IF
		END_IF

	(* set Reference Point *)
	1:	bMapInOutputs	:=TRUE;
		(*realization of a rising edge to set a nwe reference point*)
		stPZD_OUT.wCtrlW:=(ROL(stPZDOUT.wCtrlW,8))-16#1000;
		i16State		:= 2;

	2:	stPZD_OUT.wCtrlW:=(ROL(stPZDOUT.wCtrlW,8))+16#1000;
		i16State		:= 10;

	(* start home running*)
	3:	bMapInOutputs	:=TRUE;
		stPZD_OUT.PZD2	:=iCalVelo;
		(*stPZD_OUT.wCtrlW:=(ROL(stPZDOUT.wCtrlW,8))+16#800;*)
		stPZD_OUT.wCtrlW:=((ROL(stPZDOUT.wCtrlW,8)) OR 2#0000100000000000);
		icheckStatus:=2#0000010000000000;
		IF (stPZD_IN.wSTW AND icheckStatus)<>0 THEN
			(*Stophandling*)
			IF bCalibrStop THEN
				(*stPZD_OUT.wCtrlW:=(ROL(stPZDOUT.wCtrlW,8))-16#800;*)
				stPZD_OUT.wCtrlW:=((ROL(stPZDOUT.wCtrlW,8)) AND 2#1111011111111111);
				i16State	:= 10;
			ELSE
				;
			END_IF
		ELSE
			i16State:=4;
		END_IF

	4:	icheckStatus:=2#0000010000000000;
		IF ((stPZD_IN.wSTW AND icheckStatus)<>0)  THEN
			i16State	:= 10;
		END_IF
		(*Stophandling*)
		IF bCalibrStop THEN
			stPZD_OUT.wCtrlW:=(ROL(stPZDOUT.wCtrlW,8))-16#800;
			i16State	:= 10;
		END_IF

		(*Errorcase*)
	9:	bErr			:= TRUE;
		i16State		:= 10;

	10:	bbusy			:= FALSE;
		bMapInOutputs	:= FALSE;
		bSetRefPoint		:= FALSE;
		IF (NOT bSetRefPoint) AND (NOT bCalibrStart) THEN
			i16State	:= 0;
		END_IF

	END_CASE

	a_MapOutputs();
END_FUNCTION_BLOCK
ACTION a_MapInputs:
	stPZD_IN.wSTW		:=ROL(stPZDIN.wSTW,8);
	stPZD_IN.wHIW		:=ROL(stPZDIN.wHIW,8);
	stPZD_IN.PZD3		:=ROL(stPZDIN.PZD3,8);
	stPZD_IN.PZD4		:=ROL(stPZDIN.PZD4,8);
	stPZD_IN.PZD5		:=ROL(stPZDIN.PZD5,8);
	stPZD_IN.PZD6		:=ROL(stPZDIN.PZD6,8);
END_ACTION
ACTION a_MapOutputs:
IF bMapInOutputs THEN
	stPZDOUT.wCtrlW		:=ROL(stPZD_OUT.wCtrlW,8);
	stPZDOUT.PZD2		:=ROL(stPZD_OUT.PZD2,8);
	stPZDOUT.PZD3		:=ROL(stPZD_OUT.PZD3,8);
	stPZDOUT.PZD4		:=ROL(stPZD_OUT.PZD4,8);
	stPZDOUT.PZD5		:=ROL(stPZD_OUT.PZD5,8);
	stPZDOUT.PZD6		:=ROL(stPZD_OUT.PZD6,8);
END_IF
END_ACTION

(* POU FB_AX200X_Profibus, ST *)
FUNCTION_BLOCK FB_AX200X_Profibus
VAR_INPUT
	bInit					: BOOL;			(*Initialization*)
	bMode_DigitalSpeed	: BOOL;			(*OP-Mode digital speed instead of Positioning*)
	iDigitalSpeed			: DINT;			(*digital speed if OP-Mode = digital speed*)
	iVelocity				: DWORD;		(*Velocity*)
	iPosition				: DINT;			(*Position*)
	iRunningMode		: BYTE;			(*0:digital speed, 1: motiontask, 2: JogMode, 3: Calibration*)
	imotion_tasknumber	: WORD;			(*number of EEPROM-saved motion-task*)
	imotion_blocktype		: WORD:=16#2000;	(*optional Parameters of motion tasks, default:SI-values*)
	iJogModeBasicValue	: INT;			(*BasicVelocity for JogMode*)
	iCalVelo				: WORD;			(* basic velocity of Calibration*)
	bSetRefPoint			: BOOL;			(* set Reference Point*)
	bStart					: BOOL;			(*START*)
	bStop					: BOOL;			(*STOP*)
	bShortStop			: BOOL;			(* break of motion task*)
	iSlaveAddress			: BYTE;			(* Station Address of the Slave *)
	iFC310xDeviceId 		: WORD;			(* Device-ID of the FCxxxx *)
	bErrorResume		: BOOL;			(*Error resume*)
	tTimeOut				: TIME := DEFAULT_ADS_TIMEOUT;
END_VAR
VAR_OUTPUT

	bBusy				: BOOL;
	bError				: BOOL;			(*Errorstatus of Servo*)
	iErrID				: DWORD;
	bTimeOutErr		: BOOL;
	bInitOK			: BOOL;				(*Initialization OK*)
	iactPosition		 : DINT;		(*actual Position SI-value*)
END_VAR
VAR_IN_OUT
	stPZD_IN:			ST_PZD_IN;				(*Data from NC*)
	stPZD_OUT:			ST_PZD_OUT;			(*Data to NC*)
END_VAR
VAR
	istate					:INT;
	TimerPosition				:TON;
	fbAX2000_AXACT			: FB_AX2000_AXACT;
	fbAX2000_Parameter		: FB_AX2000_Parameter;
	fbAX2000_JogMode		: FB_AX2000_JogMode;
	fbAX2000_Reference		: FB_AX2000_Reference;

	iOPMode				:DWORD;
END_VAR
VAR CONSTANT
	(*Errors*)
	ERR_OPMODE	:DWORD:=1;

END_VAR
		fbAX2000_AXACT(bMode_DigitalSpeed	:=bMode_DigitalSpeed,
						iDigitalSpeed			:=iDigitalSpeed,
						iVelocity				:=iVelocity,
						 iPosition				:=iPosition ,
						 imotion_tasknumber	:=imotion_tasknumber ,
						 imotion_blocktype	:=imotion_blocktype ,
						bShortStop			:=bShortStop,
						 bErrorResume		:=bErrorResume ,
						 tTimeOut			:=tTimeOut ,
						stPZDIN				:= stPZD_IN,
						stPZDOUT			:=stPZD_OUT);
	IF iRunningMode<2 OR bInit THEN
			fbAX2000_AXACT.bStart	:=bStart;
	END_IF

	IF (NOT bInit) THEN
		fbAX2000_AXACT.bStop	:=bStop;
	END_IF

	IF fbAX2000_AXACT.stPZD_IN.wSTW =0 THEN
		bInitOK	:=FALSE;
	END_IF

	CASE istate OF

	(*action-mode*)
	0:	(*Initialization*)
		IF bInit THEN
			bBusy		:=TRUE;
			bError		:=FALSE;
			bTimeOutErr	:=FALSE;
			iErrID		:=0;
			bInitOK		:=FALSE;
			IF bMode_DigitalSpeed THEN
				iOPMode	:= 1;
			ELSE
				iOPMode	:= 2;
			END_IF
			istate		:=1;
		(*JogMode*)
		ELSIF iRunningMode=2 AND bStart THEN
			IF bInitOK THEN
				bBusy		:=TRUE;
				bError		:=FALSE;
				bTimeOutErr	:=FALSE;
				iErrID		:=0;
				istate		:=20;
			ELSE
				iErrID	:=ERR_OPMODE;
				istate	:=100;
			END_IF
		(*CalibrationMode*)
		ELSIF iRunningMode=3 AND (bStart OR  bSetRefPoint)THEN
			IF bInitOK THEN
				bBusy		:=TRUE;
				bError		:=FALSE;
				bTimeOutErr	:=FALSE;
				iErrID		:=0;
				istate		:=30;
			ELSE
				iErrID	:=ERR_OPMODE;
				istate	:=100;
			END_IF
		(*motion-task start*)
		ELSIF (iRunningMode=1 OR iRunningMode=0) AND bStart  THEN
			IF bInitOK THEN
				bBusy		:=TRUE;
				bError		:=FALSE;
				bTimeOutErr	:=FALSE;
				iErrID		:=0;
				istate		:=10;
			ELSE
				iErrID	:=ERR_OPMODE;
				istate	:=100;
			END_IF
		ELSIF iRunningMode>3 AND bStart  THEN
			iErrID	:=ERR_OPMODE;
			istate	:=100;
		END_IF

	(*Init*)
	1:	fbAX2000_AXACT.bStop	:=TRUE;
		istate	:=2;

	2:	fbAX2000_Parameter(iSlaveAddress:= iSlaveAddress,
						iPnu:= 930,
						iParameterValue:= iOPMode,
						iFC310xDeviceId:=iFC310xDeviceId ,
						bStartWrite:= TRUE );
		istate	:=3;

	3:	fbAX2000_Parameter();
		IF (NOT fbAX2000_Parameter.bBusy) THEN
			IF fbAX2000_Parameter.iErrorId<>0 THEN
				iErrID	:=fbAX2000_Parameter.iErrorId;
				bInit		:=FALSE;
				istate	:=100;
			ELSE
				istate	:=4;
			END_IF
			fbAX2000_AXACT.bStop	:=FALSE;
		END_IF

	4:	fbAX2000_Parameter(iSlaveAddress:= iSlaveAddress,
						iPnu:= 930,
						iFC310xDeviceId:=iFC310xDeviceId ,
						bStartRead:= TRUE );
		istate	:=5;

	5:	fbAX2000_Parameter();
		IF (NOT fbAX2000_Parameter.bBusy)  THEN
			IF fbAX2000_Parameter.iErrorId<>0 THEN
				iErrID	:=fbAX2000_Parameter.iErrorId;
				istate	:=100;
			ELSE
				bInitOK	:=TRUE;
				istate	:=110;
			END_IF
			bInit		:=FALSE;
		END_IF

	(*motion task start*)
	10:	IF fbAX2000_AXACT.bBusy THEN
			istate	:=11;
		ELSIF fbAX2000_AXACT.bError THEN
			fbAX2000_Parameter(iSlaveAddress:= iSlaveAddress,
							iPnu:= 1001,
							iFC310xDeviceId:=iFC310xDeviceId ,
							bStartRead:= TRUE );
			iErrID	:=fbAX2000_Parameter.iReadValue;
			istate	:=100;
		ELSIF fbAX2000_AXACT.bTimeOutErr  THEN
			bTimeOutErr	:=TRUE;
			istate	:=100;
		END_IF

	11:	fbAX2000_Parameter(iSlaveAddress:= iSlaveAddress,
						iPnu:= 1403,
						iFC310xDeviceId:=iFC310xDeviceId ,
						bStartRead:= TRUE);
		iactPosition	:=fbAX2000_Parameter.iReadValue;
		IF (NOT fbAX2000_AXACT.bBusy) THEN
			TimerPosition(in:=TRUE, PT:=t#1s);
			IF TimerPosition.Q THEN
				TimerPosition(in:=FALSE);
				istate	:=12;
			END_IF
		END_IF

	12:	fbAX2000_Parameter();
		iactPosition	:=fbAX2000_Parameter.iReadValue;
		IF (NOT fbAX2000_Parameter.bBusy) THEN
			istate	:=110;
		END_IF

	(*JogMode*)
	20:	fbAX2000_JogMode(bStart:= bStart,
						bStop		:= bStop,
						 iBasicVelo	:=iJogModeBasicValue,
						 tTimeOut	:=tTimeOut ,
						stPZDIN		:= stPZD_IN,
						stPZDOUT	:=stPZD_OUT);
		fbAX2000_Parameter(iSlaveAddress:= iSlaveAddress,
						iPnu:= 1403,
						iFC310xDeviceId:=iFC310xDeviceId ,
						bStartRead:= TRUE);
		iactPosition	:=fbAX2000_Parameter.iReadValue;
		IF bStop OR fbAX2000_JogMode.bErr OR fbAX2000_JogMode.bTimeOutErr THEN
			istate	:=21;
		END_IF

	21:	fbAX2000_Parameter();
		iactPosition	:=fbAX2000_Parameter.iReadValue;
		IF (NOT fbAX2000_Parameter.bBusy) THEN
			bStart		:= FALSE;
			fbAX2000_JogMode(bStart		:= bStart,
							bStop		:= FALSE,
							 iBasicVelo	:=iJogModeBasicValue,
							 tTimeOut	:=tTimeOut ,
							stPZDIN		:= stPZD_IN,
							stPZDOUT	:=stPZD_OUT);
			istate	:=110;
			IF fbAX2000_JogMode.bErr THEN
				fbAX2000_Parameter(iSlaveAddress:= iSlaveAddress,
								iPnu:= 1001,
								iFC310xDeviceId:=iFC310xDeviceId ,
								bStartRead:= TRUE );
				iErrID	:=fbAX2000_Parameter.iReadValue;
				istate	:=100;
			ELSIF fbAX2000_JogMode.bTimeOutErr THEN
				bTimeOutErr	:=TRUE;
			END_IF
		END_IF

	(*CalibrationMode*)
	30:	fbAX2000_Reference(bSetRefPoint	:= bSetRefPoint ,
						bCalibrStart		:= bStart,
						bCalibrStop		:= bStop,
						iCalVelo			:= iCalVelo,
						stPZDIN			:= stPZD_IN,
						stPZDOUT		:=stPZD_OUT);
		fbAX2000_Parameter(iSlaveAddress:= iSlaveAddress,
						iPnu:= 1403,
						iFC310xDeviceId:=iFC310xDeviceId ,
						bStartRead:= TRUE);
		iactPosition	:=fbAX2000_Parameter.iReadValue;
		IF bStop OR fbAX2000_Reference.bErr  THEN
			istate	:=31;
		END_IF

	31:	fbAX2000_Parameter();
		iactPosition	:=fbAX2000_Parameter.iReadValue;
		IF (NOT fbAX2000_Parameter.bBusy) THEN
			bStart		:= FALSE;
			fbAX2000_Reference(bCalibrStart	:= bStart,
							bCalibrStop		:= TRUE,
							stPZDIN			:= stPZD_IN,
							stPZDOUT		:=stPZD_OUT);
			istate	:=110;
			IF fbAX2000_Reference.bErr THEN
				fbAX2000_Parameter(iSlaveAddress:= iSlaveAddress,
								iPnu:= 1001,
								iFC310xDeviceId:=iFC310xDeviceId ,
								bStartRead:= TRUE );
				iErrID	:=fbAX2000_Parameter.iReadValue;
				istate	:=100;
			END_IF
		END_IF


	(*Error*)
	100:	bError	:=TRUE;
		istate	:=110;

	(*Quit*)
	110:	bBusy	:=FALSE;
		IF (NOT bStart) AND (NOT bInit) THEN
			istate	:=0;
		END_IF


	ELSE
		;
	END_CASE
END_FUNCTION_BLOCK

(* POU FB_Dpv1Read, ST *)
FUNCTION_BLOCK FB_Dpv1Read
(*****************************************************************************************************************
	DESCRIPTION:	This FUNCTION block implements DPV1 Parameter Read

	CHANGE LOG:
	BY		DATE		DESCRIPTION OF CHANGE
	ICh		2016/06/02	adjustable delay via global tCommDelayDPV1 (default for 100ms)
	ICh		2008/04/02	delay resend request after fault for 100ms
	ICh		2007/01/08	resend request after fault
	ICh		2007/01/05	iRequestRef limited to 128
	ICh		2006/08/09	wait timer decreased, bugfix for errors
	ICh		2006/07/12	Bugfix iRequestRef as VAR_IN_OUT
	ICh		2006/07/10	Bugfix for evaluate response; enhanced error reporting
	ICh		2006/07/05	First Version

******************************************************************************************************************)
VAR_INPUT
	bExecute			: BOOL;

	(* drive access info *)
	aNetId				: T_AmsNetId;	(* NetID of Profibus Master FC310x/EL6731 *)
	iProfibusSlaveAdr	: USINT;	 	(* DP address of ProfiDrive *)
	iDriveId			: USINT;		(* 0..255 possible *)
	pDpv1ReqData		: POINTER TO ARRAY [1..iMAX_DPV1_SIZE] OF BYTE;
	iDpv1ReqDataLen		: UDINT;
	pDpv1ResData		: POINTER TO ARRAY [1..iMAX_DPV1_SIZE] OF BYTE;
	iDpv1ResDataLen		: UDINT;
	tTmOut				: TIME := DEFAULT_ADS_TIMEOUT;
END_VAR
VAR_OUTPUT
	bBusy				: BOOL;
	bError				: BOOL;
	bErrorValues		: BOOL;
	iErrId				: UDINT;
	iErrorClass			: BYTE;
	iErrorCode			: BYTE;
END_VAR
VAR_IN_OUT
	iRequestRef			: USINT;		(* 1..127;    0: reserved *)
END_VAR
VAR
	fbWriteAccessData 	: ADSWRITE;
	fbReadData 			: ADSREAD;
	iState				: INT;
	bExecute_			: BOOL;

	stDpv1ReqHeader		: ST_Dpv1Header;
	stDpv1ResHeader		: ST_Dpv1Header;

	WaitTimer			: TON := (PT := T#100ms);
	TmOutTimer			: TON;
END_VAR
TmOutTimer();

CASE iState OF
0:	(* idle until rising edge on bExecute *)
	IF bExecute AND NOT bExecute_ THEN
		(* generate request reference *)
		iRequestRef := UINT_TO_USINT((USINT_TO_UINT(iRequestRef) + 1) MOD 128);
		IF iRequestRef = 0 THEN
			iRequestRef := 1;
		END_IF
		pDpv1ReqData^[1] := iRequestRef;
		MEMCPY(ADR(stDpv1ReqHeader), pDpv1ReqData, SIZEOF(stDpv1ReqHeader));

		(* clear response data *)
		MEMSET(pDpv1ResData, 0, iMAX_DPV1_SIZE);

		(* on rising edge *)
		bExecute_ 	:= bExecute;
		bBusy		:= TRUE;
		bError		:= FALSE;
		bErrorValues:= FALSE;
		iErrId		:= 0;
		iErrorClass	:= 0;
		iErrorCode	:= 0;

		(* complete read request timeout 12 times the ADS timeout *)
		TmOutTimer(IN := FALSE, PT := MAX(tTmOut * 12, T#30s));
		TmOutTimer(IN := TRUE);

		(* send request *)
		fbWriteAccessData(
			NETID	:= aNetId,
			PORT	:= 16#1000 + iProfibusSlaveAdr,
			IDXGRP	:= 0,
			IDXOFFS	:= 47,
			LEN		:= MIN(iDpv1ReqDataLen, iMAX_DPV1_SIZE),
			SRCADDR	:= pDpv1ReqData,
			WRITE	:= FALSE,
			TMOUT	:= tTmOut
		);
		fbWriteAccessData(WRITE	:= TRUE);

		iState := 1;
	END_IF

1:	(* write access data for DPV1 read request *)
	fbWriteAccessData(WRITE	:= FALSE);

	IF NOT fbWriteAccessData.BUSY THEN
		fbWriteAccessData(WRITE	:= FALSE);

		IF NOT fbWriteAccessData.ERR THEN
			(* read request parameter successfully sent, check for response *)
			WaitTimer(IN := FALSE);
			iState	:= 2; (* wait before polling *)
		ELSE
			bBusy	:= FALSE;
			bError	:= TRUE;
			iErrId	:= fbWriteAccessData.ERRID;
			IF ((UDINT_TO_DWORD(iErrId) AND DWORD#16#FF000000) = DWORD#16#27000000) THEN
				iErrorClass := UDINT_TO_BYTE(SHR((UDINT_TO_DWORD(iErrId) AND 16#00F00000), 20));
				iErrorCode := UDINT_TO_BYTE(SHR((UDINT_TO_DWORD(iErrId) AND 16#000F0000), 16));
			END_IF
			iState	:= 0;
		END_IF
	END_IF

2:	(* wait staate before next read response check *)
	WaitTimer(IN := TRUE, PT := tCommDelayDPV1);
	IF WaitTimer.Q THEN
		(* read request parameter successfully sent, check for read response *)
		MEMSET(pDpv1ResData, 0, iMAX_DPV1_SIZE);
		fbReadData(
			NETID	:= aNetId,
			PORT	:= 16#1000 + iProfibusSlaveAdr,
			IDXGRP	:= 0,
			IDXOFFS	:= 47,
			LEN		:= iMAX_DPV1_SIZE,
			DESTADDR:= pDpv1ResData,
			READ	:= FALSE,
			TMOUT	:= tTmOut,
		);
		fbReadData(READ := TRUE);
		iState	:= 3; (* CHECK READ *)
	END_IF

3:	(* wait for read response with data from DPV1 read request *)
	fbReadData(READ := FALSE);

	IF NOT fbReadData.BUSY THEN
		fbReadData(READ := FALSE);
		IF NOT fbReadData.ERR THEN
			MEMCPY(ADR(stDpv1ResHeader), pDpv1ResData, SIZEOF(stDpv1ResHeader));

			(* check for read response reference *)
			IF (stDpv1ResHeader.iRequestRef = stDpv1ReqHeader.iRequestRef) AND (stDpv1ResHeader.iAxis = stDpv1ReqHeader.iAxis) THEN
				(* response to last parameter request - split response data *)
				TmOutTimer(IN := FALSE);
				iState	:= 5;	(* DONE *)
			ELSIF stDpv1ResHeader.iRequestRef = 0 THEN
				(* no response *)
				IF TmOutTimer.Q THEN
					(* complete read request timed out *)
					TmOutTimer(IN := FALSE);
					bBusy	:= FALSE;
					bError	:= TRUE;
					iErrId	:= 16#745; (* timeout *)
					iState	:= 0; (* ERROR *)
				ELSE
					(* no response, go to wait state *)
					WaitTimer(IN := FALSE);
					iState	:= 2; (* WAIT and REPEAT *)
				END_IF
			ELSE
				(* wrong response *)
				bBusy	:= FALSE;
				bError	:= TRUE;
				iErrId	:= 2; (* wrong reference response *)
				iState	:= 0; (* ERROR *)
			END_IF
		ELSE
			IF ((UDINT_TO_DWORD(fbReadData.ERRID) AND DWORD#16#FFFF0000) = DWORD#16#27B50000) THEN
				(* repeat telegram *)
				WaitTimer(IN := FALSE);
				iState	:= 4; (* SEND NEW REQUEST *)
			ELSE
				(* error *)
				bBusy	:= FALSE;
				bError	:= TRUE;
				iErrId	:= fbReadData.ERRID;
				IF ((UDINT_TO_DWORD(iErrId) AND DWORD#16#FF000000) = DWORD#16#27000000) THEN
					iErrorClass := UDINT_TO_BYTE(SHR((UDINT_TO_DWORD(iErrId) AND 16#00F00000), 20));
					iErrorCode := UDINT_TO_BYTE(SHR((UDINT_TO_DWORD(iErrId) AND 16#000F0000), 16));
				END_IF
				iState	:= 0; (* ERROR *)
			END_IF
		END_IF
	END_IF

4:	(* generate new request reference after fault *)
	WaitTimer(IN := TRUE, PT := tCommDelayDPV1);
	IF WaitTimer.Q THEN
		iRequestRef := UINT_TO_USINT((USINT_TO_UINT(iRequestRef) + 1) MOD 128);
		IF iRequestRef = 0 THEN
			iRequestRef := 1;
		END_IF
		pDpv1ReqData^[1] := iRequestRef;
		MEMCPY(ADR(stDpv1ReqHeader), pDpv1ReqData, SIZEOF(stDpv1ReqHeader));
	
		(* clear response data *)
		MEMSET(pDpv1ResData, 0, iMAX_DPV1_SIZE);
	
		(* send request *)
		fbWriteAccessData(
			NETID	:= aNetId,
			PORT	:= 16#1000 + iProfibusSlaveAdr,
			IDXGRP	:= 0,
			IDXOFFS	:= 47,
			LEN		:= MIN(iDpv1ReqDataLen, iMAX_DPV1_SIZE),
			SRCADDR	:= pDpv1ReqData,
			WRITE	:= FALSE,
			TMOUT	:= tTmOut
		);
		fbWriteAccessData(WRITE	:= TRUE);
	
		iState := 1; (* CHECK WRITE *)
	END_IF

5:	(* evaluate response *)
	IF stDpv1ResHeader.iRequestID = stDpv1ReqHeader.iRequestID THEN
		(* DPV1 Read successful - done *)
		bBusy	:= FALSE;
		iState	:= 0; (* DONE *)
	ELSIF (SINT_TO_BYTE(stDpv1ResHeader.iRequestID) AND 16#7F) = SINT_TO_BYTE(stDpv1ReqHeader.iRequestID) THEN
		(* DPV1 Read not successful or partly not successful *)
		bErrorValues:= TRUE;
		bBusy	:= FALSE;
		bError	:= TRUE;
		iErrId	:= 3; (* DPV1 Read not successful or partly not successful *)
		iState	:= 0; (* ERROR *)
	ELSE
		(* wrong response *)
		bBusy	:= FALSE;
		bError	:= TRUE;
		iErrId	:= 4; (* wrong response ID *)
		iState	:= 0; (* ERROR *)
	END_IF

END_CASE

(* clear flag *)
bExecute_ := bExecute_ AND bExecute;
END_FUNCTION_BLOCK

(* POU FB_Dpv1ReadPNET, ST *)
FUNCTION_BLOCK FB_Dpv1ReadPNET
(*****************************************************************************************************************
	DESCRIPTION:	This FUNCTION block implements DPV1 Parameter Read for Profinet

	CHANGE LOG:
	BY		DATE		DESCRIPTION OF CHANGE
	ICh		2009/07/23	First Version
	ICh		2016/02/17	repeat read response instead of new write request in case of busy response
	ICh		2016/06/02	adjustable delay via global tCommDelayDPV1PNET (default for 100ms)

******************************************************************************************************************)
VAR_INPUT
	bExecute			: BOOL;

	(* drive access info *)
	aNetId				: T_AmsNetId;	(* NetID of Profibus Master EL6631 *)
	iProfinetPort		: UINT;		 	(* Port of ProfiDrive *)
	iDriveId			: USINT;		(* 0..255 possible *)
	pDpv1ReqData		: POINTER TO ARRAY [1..iMAX_DPV1_SIZE_PNET_REQ] OF BYTE;
	iDpv1ReqDataLen		: UDINT;
	pDpv1ResData		: POINTER TO ARRAY [1..iMAX_DPV1_SIZE_PNET_RES] OF BYTE;
	iDpv1ResDataLen		: UDINT;
	tTmOut				: TIME;
END_VAR
VAR_OUTPUT
	bBusy				: BOOL;
	bError				: BOOL;
	bErrorValues		: BOOL;
	iErrId				: UDINT;
	iErrorClass			: BYTE;
	iErrorCode			: BYTE;
END_VAR
VAR_IN_OUT
	iRequestRef			: USINT;		(* 1..127;    0: reserved *)
END_VAR
VAR
	fbRWData 			: ADSRDWRT;
	iState				: INT;
	bExecute_			: BOOL;
	iIGrp				: UDINT := 16#F823;
	stDpv1ReqHeader		: ST_Dpv1Header;
	stDpv1ResHeader		: ST_Dpv1Header;
	stPNETFrameHeader	: ST_PNIOConfigRecord;

	WaitTimer			: TON := (PT := T#100ms);
	TmOutTimer			: TON;
END_VAR
TmOutTimer();

CASE iState OF
0:	(* idle until rising edge on bExecute *)
	IF bExecute AND NOT bExecute_ THEN
		(* generate request reference *)
		iRequestRef := UINT_TO_USINT((USINT_TO_UINT(iRequestRef) + 1) MOD 128);
		IF iRequestRef = 0 THEN
			iRequestRef := 1;
		END_IF
		pDpv1ReqData^[1] := 1; pDpv1ReqData^[2] := 0; (* write request *)
		pDpv1ReqData^[1+SIZEOF(stPNETFrameHeader)] := iRequestRef;
		MEMCPY(ADR(stPNETFrameHeader), pDpv1ReqData, SIZEOF(stPNETFrameHeader));
		MEMCPY(ADR(stDpv1ReqHeader), pDpv1ReqData+SIZEOF(stPNETFrameHeader), SIZEOF(stDpv1ReqHeader));

		(* clear response data *)
		MEMSET(pDpv1ResData, 0, iMAX_DPV1_SIZE_PNET_RES);

		(* on rising edge *)
		bExecute_ 	:= bExecute;
		bBusy		:= TRUE;
		bError		:= FALSE;
		bErrorValues:= FALSE;
		iErrId		:= 0;
		iErrorClass	:= 0;
		iErrorCode	:= 0;

		(* complete request timeout *)
		TmOutTimer(IN := FALSE, PT := LIMIT(T#5s, INT_TO_TIME(INT#12*TIME_TO_INT(tTmOut)), T#60s));
		TmOutTimer(IN := TRUE);

		(* send request *)
		fbRWData(
			NETID	:= aNetId,
			PORT	:= iProfinetPort,
			IDXGRP	:= iIGrp,
			IDXOFFS	:= 0,
			WRITELEN:= MIN(iDpv1ReqDataLen, iMAX_DPV1_SIZE_PNET_REQ),
			SRCADDR	:= pDpv1ReqData,
			READLEN	:= MIN(iDpv1ResDataLen, iMAX_DPV1_SIZE_PNET_RES),
			DESTADDR:= pDpv1ResData,
			WRTRD	:= FALSE,
			TMOUT	:= tTmOut
		);
		fbRWData(WRTRD	:= TRUE);
		iState := 1;
	END_IF

1:	(* write access data for DPV1 read request *)
	fbRWData(WRTRD	:= FALSE);

	IF NOT fbRWData.BUSY THEN
		fbRWData(WRTRD	:= FALSE);

		IF NOT fbRWData.ERR THEN
			(* read request parameter successfully sent, check for response *)
			WaitTimer(IN := FALSE);
			iState	:= 2; (* wait before polling *)
		ELSE
			bBusy	:= FALSE;
			bError	:= TRUE;
			iErrId	:= fbRWData.ERRID;
			IF ((UDINT_TO_DWORD(iErrId) AND DWORD#16#FF000000) = DWORD#16#27000000) THEN
				iErrorClass := UDINT_TO_BYTE(SHR((UDINT_TO_DWORD(iErrId) AND 16#00F00000), 20));
				iErrorCode := UDINT_TO_BYTE(SHR((UDINT_TO_DWORD(iErrId) AND 16#000F0000), 16));
			END_IF
			iState	:= 0;
		END_IF
	END_IF

2:	(* wait staate before next read response check *)
	WaitTimer(IN := TRUE, PT := tCommDelayDPV1PNET);
	IF WaitTimer.Q THEN
		stPNETFrameHeader.iRW := 0; (* read response *)
		stPNETFrameHeader.stPNIORecord.iLength := UDINT_TO_INT(MIN(iDpv1ResDataLen, iMAX_DPV1_SIZE_PNET_RES)); (* max read response length *)

		(* read request parameter successfully sent, check for read response *)
		MEMSET(pDpv1ResData, 0, iMAX_DPV1_SIZE_PNET_RES);
		fbRWData(
			NETID	:= aNetId,
			PORT	:= iProfinetPort,
			IDXGRP	:= iIGrp,
			IDXOFFS	:= 0,
			WRITELEN:= SIZEOF(stPNETFrameHeader),
			SRCADDR	:= ADR(stPNETFrameHeader),
			READLEN	:= MIN(iDpv1ResDataLen, iMAX_DPV1_SIZE_PNET_RES),
			DESTADDR:= pDpv1ResData,
			WRTRD	:= FALSE,
			TMOUT	:= tTmOut
		);
		fbRWData(WRTRD	:= TRUE);
		iState	:= 3; (* CHECK READ *)
	END_IF

3:	(* wait for read response with data from DPV1 read request *)
	fbRWData(WRTRD	:= FALSE);

	IF NOT fbRWData.BUSY THEN
		fbRWData(WRTRD := FALSE);
		IF NOT fbRWData.ERR THEN
			MEMCPY(ADR(stDpv1ResHeader), pDpv1ResData, SIZEOF(stDpv1ResHeader));

			(* check for read response reference *)
			IF (stDpv1ResHeader.iRequestRef = stDpv1ReqHeader.iRequestRef) AND (stDpv1ResHeader.iAxis = stDpv1ReqHeader.iAxis) THEN
				(* response to last parameter request - split response data *)
				TmOutTimer(IN := FALSE);
				iState	:= 4;	(* DONE *)
			ELSIF stDpv1ResHeader.iRequestRef = 0 THEN
				(* no response *)
				IF TmOutTimer.Q THEN
					(* complete read request timed out *)
					TmOutTimer(IN := FALSE);
					bBusy	:= FALSE;
					bError	:= TRUE;
					iErrId	:= 16#745; (* timeout *)
					iState	:= 0; (* ERROR *)
				ELSE
					(* no response, go to wait state *)
					WaitTimer(IN := FALSE);
					iState	:= 2; (* WAIT and REPEAT *)
				END_IF
			ELSE
				(* wrong response *)
				bBusy	:= FALSE;
				bError	:= TRUE;
				iErrId	:= 2; (* wrong reference response *)
				iState	:= 0; (* ERROR *)
			END_IF
		ELSE
			IF ((UDINT_TO_DWORD(fbRWData.ERRID) AND DWORD#16#FFFF0000) = DWORD#16#27B50000) OR ((UDINT_TO_DWORD(fbRWData.ERRID) AND DWORD#16#0000FFFF) = DWORD#16#00000723) THEN
				(* no response *)
				IF TmOutTimer.Q THEN
					(* complete read request timed out *)
					TmOutTimer(IN := FALSE);
					bBusy	:= FALSE;
					bError	:= TRUE;
					iErrId	:= 16#745; (* timeout *)
					iState	:= 0; (* ERROR *)
				ELSE
					(* no response, go to wait state *)
					WaitTimer(IN := FALSE);
					iState	:= 2; (* WAIT and REPEAT *)
				END_IF
			ELSE
				(* error *)
				bBusy	:= FALSE;
				bError	:= TRUE;
				iErrId	:= fbRWData.ERRID;
				IF ((UDINT_TO_DWORD(iErrId) AND DWORD#16#FF000000) = DWORD#16#27000000) THEN
					iErrorClass := UDINT_TO_BYTE(SHR((UDINT_TO_DWORD(iErrId) AND 16#00F00000), 20));
					iErrorCode := UDINT_TO_BYTE(SHR((UDINT_TO_DWORD(iErrId) AND 16#000F0000), 16));
				END_IF
				iState	:= 0; (* ERROR *)
			END_IF
		END_IF
	END_IF

4:	(* evaluate response *)
	IF stDpv1ResHeader.iRequestID = stDpv1ReqHeader.iRequestID THEN
		(* DPV1 Read successful - done *)
		bBusy	:= FALSE;
		iState	:= 0; (* DONE *)
	ELSIF (SINT_TO_BYTE(stDpv1ResHeader.iRequestID) AND 16#7F) = SINT_TO_BYTE(stDpv1ReqHeader.iRequestID) THEN
		(* DPV1 Read not successful or partly not successful *)
		bErrorValues:= TRUE;
		bBusy	:= FALSE;
		bError	:= TRUE;
		iErrId	:= 3; (* DPV1 Read not successful or partly not successful *)
		iState	:= 0; (* ERROR *)
	ELSE
		(* wrong response *)
		bBusy	:= FALSE;
		bError	:= TRUE;
		iErrId	:= 4; (* wrong response ID *)
		iState	:= 0; (* ERROR *)
	END_IF

END_CASE

(* clear flag *)
bExecute_ := bExecute_ AND bExecute;
END_FUNCTION_BLOCK

(* POU FB_Dpv1Write, ST *)
FUNCTION_BLOCK FB_Dpv1Write
(*****************************************************************************************************************
	DESCRIPTION:	This FUNCTION block implements DPV1 Parameter Write

	CHANGE LOG:
	BY		DATE		DESCRIPTION OF CHANGE
	ICh		2016/06/02	adjustable delay via global tCommDelayDPV1 (default for 100ms)
	ICh		2008/04/02	delay resend request after fault for 100ms
	ICh		2007/01/08	resend request after fault
	ICh		2007/01/05	iRequestRef limited to 128
	ICh		2006/08/09	wait timer decreased, bugfix for errors
	ICh		2006/07/12	Bugfix iRequestRef as VAR_IN_OUT
	ICh		2006/07/10	Bugfix for evaluate response; enhanced error reporting
	ICh		2006/07/07	First Version

******************************************************************************************************************)
VAR_INPUT
	bExecute			: BOOL;

	(* drive access info *)
	aNetId				: T_AmsNetId;	(* NetID of Profibus Master FC310x/EL6731 *)
	iProfibusSlaveAdr	: USINT;	 	(* DP address of ProfiDrive *)
	iDriveId			: USINT;		(* 0..255 possible *)
	pDpv1ReqData		: POINTER TO ARRAY [1..iMAX_DPV1_SIZE] OF BYTE;
	iDpv1ReqDataLen		: UDINT;
	pDpv1ResData		: POINTER TO ARRAY [1..iMAX_DPV1_SIZE] OF BYTE;
	iDpv1ResDataLen		: UDINT;
	tTmOut				: TIME := DEFAULT_ADS_TIMEOUT;
END_VAR
VAR_OUTPUT
	bBusy				: BOOL;
	bError				: BOOL;
	bErrorValues		: BOOL;
	iErrId				: UDINT;
	iErrorClass			: BYTE;
	iErrorCode			: BYTE;
END_VAR
VAR_IN_OUT
	iRequestRef			: USINT;		(* 1..127;    0: reserved *)
END_VAR
VAR
	fbWriteAccessData 	: ADSWRITE;
	fbReadData 			: ADSREAD;
	iState				: INT;
	bExecute_			: BOOL;

	stDpv1ReqHeader		: ST_Dpv1Header;
	stDpv1ResHeader		: ST_Dpv1Header;

	WaitTimer			: TON := (PT := T#100ms);
	TmOutTimer			: TON;
END_VAR
TmOutTimer();

CASE iState OF
0:	(* idle until rising edge on bExecute *)
	IF bExecute AND NOT bExecute_ THEN
		(* generate request reference *)
		iRequestRef := UINT_TO_USINT((USINT_TO_UINT(iRequestRef) + 1) MOD 128);
		IF iRequestRef = 0 THEN
			iRequestRef := 1;
		END_IF
		pDpv1ReqData^[1] := iRequestRef;
		MEMCPY(ADR(stDpv1ReqHeader), pDpv1ReqData, SIZEOF(stDpv1ReqHeader));

		(* clear response data *)
		MEMSET(pDpv1ResData, 0, iMAX_DPV1_SIZE);

		(* on rising edge *)
		bExecute_ 	:= bExecute;
		bBusy		:= TRUE;
		bError		:= FALSE;
		bErrorValues:= FALSE;
		iErrId		:= 0;
		iErrorClass	:= 0;
		iErrorCode	:= 0;

		(* complete read request timeout 12 times the ADS timeout *)
		TmOutTimer(IN := FALSE, PT := MAX(tTmOut * 12, T#30s));
		TmOutTimer(IN := TRUE);

		(* send request *)
		fbWriteAccessData(
			NETID	:= aNetId,
			PORT	:= 16#1000 + iProfibusSlaveAdr,
			IDXGRP	:= 0,
			IDXOFFS	:= 47,
			LEN		:= MIN(iDpv1ReqDataLen, iMAX_DPV1_SIZE),
			SRCADDR	:= pDpv1ReqData,
			WRITE	:= FALSE,
			TMOUT	:= tTmOut
		);
		fbWriteAccessData(WRITE	:= TRUE);

		iState := 1;
	END_IF

1:	(* write access data for DPV1 read request *)
	fbWriteAccessData(WRITE	:= FALSE);

	IF NOT fbWriteAccessData.BUSY THEN
		fbWriteAccessData(WRITE	:= FALSE);

		IF NOT fbWriteAccessData.ERR THEN
			(* read request parameter successfully sent, check for response *)
			WaitTimer(IN := FALSE);
			iState	:= 2; (* wait before polling *)
		ELSE
			bBusy	:= FALSE;
			bError	:= TRUE;
			iErrId	:= fbWriteAccessData.ERRID;
			IF ((UDINT_TO_DWORD(iErrId) AND DWORD#16#FF000000) = DWORD#16#27000000) THEN
				iErrorClass := UDINT_TO_BYTE(SHR((UDINT_TO_DWORD(iErrId) AND 16#00F00000), 20));
				iErrorCode := UDINT_TO_BYTE(SHR((UDINT_TO_DWORD(iErrId) AND 16#000F0000), 16));
			END_IF
			iState	:= 0;
		END_IF
	END_IF

2:	(* wait staate before next read response check *)
	WaitTimer(IN := TRUE, PT := tCommDelayDPV1);
	IF WaitTimer.Q THEN
		(* read request parameter successfully sent, check for read response *)
		MEMSET(pDpv1ResData, 0, iMAX_DPV1_SIZE);
		fbReadData(
			NETID	:= aNetId,
			PORT	:= 16#1000 + iProfibusSlaveAdr,
			IDXGRP	:= 0,
			IDXOFFS	:= 47,
			LEN		:= iMAX_DPV1_SIZE,
			DESTADDR:= pDpv1ResData,
			READ	:= FALSE,
			TMOUT	:= tTmOut,
		);
		fbReadData(READ := TRUE);
		iState	:= 3; (* CHECK READ *)
	END_IF

3:	(* wait for read response with data from DPV1 read request *)
	fbReadData(READ := FALSE);

	IF NOT fbReadData.BUSY THEN
		fbReadData(READ := FALSE);
		IF NOT fbReadData.ERR THEN
			MEMCPY(ADR(stDpv1ResHeader), pDpv1ResData, SIZEOF(stDpv1ResHeader));

			(* check for read response reference *)
			IF (stDpv1ResHeader.iRequestRef = stDpv1ReqHeader.iRequestRef) AND (stDpv1ResHeader.iAxis = stDpv1ReqHeader.iAxis) THEN
				(* response to last parameter request - split response data *)
				TmOutTimer(IN := FALSE);
				iState	:= 5; (* DONE *)
			ELSIF stDpv1ResHeader.iRequestRef = 0 THEN
				(* no response *)
				IF TmOutTimer.Q THEN
					(* complete read request timed out *)
					TmOutTimer(IN := FALSE);
					bBusy	:= FALSE;
					bError	:= TRUE;
					iErrId	:= 16#745; (* timeout *)
					iState	:= 0; (* ERROR *)
				ELSE
					(* no response, go to wait state *)
					WaitTimer(IN := FALSE);
					iState	:= 2; (* WAIT and REPEAT *)
				END_IF
			ELSE
				(* wrong response *)
				bBusy	:= FALSE;
				bError	:= TRUE;
				iErrId	:= 2; (* wrong reference response *)
				iState	:= 0; (* ERROR *)
			END_IF
		ELSE
			IF ((UDINT_TO_DWORD(fbReadData.ERRID) AND DWORD#16#FFFF0000) = DWORD#16#27B50000) THEN
				(* repeat telegram *)
				WaitTimer(IN := FALSE);
				iState	:=  4; (* SEND NEW REQUEST *)
			ELSE
				(* error *)
				bBusy	:= FALSE;
				bError	:= TRUE;
				iErrId	:= fbReadData.ERRID;
				IF ((UDINT_TO_DWORD(iErrId) AND DWORD#16#FF000000) = DWORD#16#27000000) THEN
					iErrorClass := UDINT_TO_BYTE(SHR((UDINT_TO_DWORD(iErrId) AND 16#00F00000), 20));
					iErrorCode := UDINT_TO_BYTE(SHR((UDINT_TO_DWORD(iErrId) AND 16#000F0000), 16));
				END_IF
				iState	:= 0; (* ERROR *)
			END_IF
		END_IF
	END_IF

4:	(* generate new request reference after fault *)
	WaitTimer(IN := TRUE, PT := tCommDelayDPV1);
	IF WaitTimer.Q THEN
		iRequestRef := UINT_TO_USINT((USINT_TO_UINT(iRequestRef) + 1) MOD 128);
		IF iRequestRef = 0 THEN
			iRequestRef := 1;
		END_IF
		pDpv1ReqData^[1] := iRequestRef;
		MEMCPY(ADR(stDpv1ReqHeader), pDpv1ReqData, SIZEOF(stDpv1ReqHeader));
	
		(* clear response data *)
		MEMSET(pDpv1ResData, 0, iMAX_DPV1_SIZE);
	
		(* send request *)
		fbWriteAccessData(
			NETID	:= aNetId,
			PORT	:= 16#1000 + iProfibusSlaveAdr,
			IDXGRP	:= 0,
			IDXOFFS	:= 47,
			LEN		:= MIN(iDpv1ReqDataLen, iMAX_DPV1_SIZE),
			SRCADDR	:= pDpv1ReqData,
			WRITE	:= FALSE,
			TMOUT	:= tTmOut
		);
		fbWriteAccessData(WRITE	:= TRUE);
	
		iState := 1; (* CHECK WRITE *)
	END_IF

5:	(* evaluate response *)
	IF stDpv1ResHeader.iRequestID = stDpv1ReqHeader.iRequestID THEN
		(* DPV1 Read successful - done *)
		bBusy	:= FALSE;
		iState	:= 0; (* DONE *)
	ELSIF (SINT_TO_BYTE(stDpv1ResHeader.iRequestID) AND 16#7F) = SINT_TO_BYTE(stDpv1ReqHeader.iRequestID) THEN
		(* DPV1 Read not successful or partly not successful *)
		bErrorValues:= TRUE;
		bBusy	:= FALSE;
		bError	:= TRUE;
		iErrId	:= 3; (* DPV1 Write not successful or partly not successful *)
		iState	:= 0; (* ERROR *)
	ELSE
		(* wrong response *)
		bBusy	:= FALSE;
		bError	:= TRUE;
		iErrId	:= 4; (* wrong response ID *)
		iState	:= 0; (* ERROR *)
	END_IF
END_CASE

(* clear flag *)
bExecute_ := bExecute_ AND bExecute;
END_FUNCTION_BLOCK

(* POU FB_Dpv1WritePNET, ST *)
FUNCTION_BLOCK FB_Dpv1WritePNET
(*****************************************************************************************************************
	DESCRIPTION:	This FUNCTION block implements DPV1 Parameter Write for Profinet

	CHANGE LOG:
	BY		DATE		DESCRIPTION OF CHANGE
	ICh		2009/07/23	First Version
	ICh		2016/02/17	repeat read response instead of new write request in case of busy response
	ICh		2016/06/02	adjustable delay via global tCommDelayDPV1PNET (default for 100ms)

******************************************************************************************************************)
VAR_INPUT
	bExecute			: BOOL;

	(* drive access info *)
	aNetId				: T_AmsNetId;	(* NetID of Profinet Master EL6631 *)
	iProfinetPort		: UINT;		 	(* Port of ProfiDrive *)
	iDriveId			: USINT;		(* 0..255 possible *)
	pDpv1ReqData		: POINTER TO ARRAY [1..iMAX_DPV1_SIZE_PNET_REQ] OF BYTE;
	iDpv1ReqDataLen		: UDINT;
	pDpv1ResData		: POINTER TO ARRAY [1..iMAX_DPV1_SIZE_PNET_RES] OF BYTE;
	iDpv1ResDataLen		: UDINT;
	tTmOut				: TIME;
END_VAR
VAR_OUTPUT
	bBusy				: BOOL;
	bError				: BOOL;
	bErrorValues		: BOOL;
	iErrId				: UDINT;
	iErrorClass			: BYTE;
	iErrorCode			: BYTE;
END_VAR
VAR_IN_OUT
	iRequestRef			: USINT;		(* 1..127;    0: reserved *)
END_VAR
VAR
	fbRWData 			: ADSRDWRT;
	iState				: INT;
	bExecute_			: BOOL;
	iIGrp				: UDINT := 16#F823;
	stDpv1ReqHeader		: ST_Dpv1Header;
	stDpv1ResHeader		: ST_Dpv1Header;
	stPNETFrameHeader	: ST_PNIOConfigRecord;

	WaitTimer			: TON := (PT := T#100ms);
	TmOutTimer			: TON;
END_VAR
TmOutTimer();

CASE iState OF
0:	(* idle until rising edge on bExecute *)
	IF bExecute AND NOT bExecute_ THEN
		(* generate request reference *)
		iRequestRef := UINT_TO_USINT((USINT_TO_UINT(iRequestRef) + 1) MOD 128);
		IF iRequestRef = 0 THEN
			iRequestRef := 1;
		END_IF
		pDpv1ReqData^[1] := 1; pDpv1ReqData^[2] := 0; (* write request *)
		pDpv1ReqData^[1+SIZEOF(stPNETFrameHeader)] := iRequestRef;
		MEMCPY(ADR(stPNETFrameHeader), pDpv1ReqData, SIZEOF(stPNETFrameHeader));
		MEMCPY(ADR(stDpv1ReqHeader), pDpv1ReqData+SIZEOF(stPNETFrameHeader), SIZEOF(stDpv1ReqHeader));

		(* clear response data *)
		MEMSET(pDpv1ResData, 0, iMAX_DPV1_SIZE_PNET_RES);

		(* on rising edge *)
		bExecute_ 	:= bExecute;
		bBusy		:= TRUE;
		bError		:= FALSE;
		bErrorValues:= FALSE;
		iErrId		:= 0;
		iErrorClass	:= 0;
		iErrorCode	:= 0;

		(* complete request timeout *)
		TmOutTimer(IN := FALSE, PT := LIMIT(T#5s, INT_TO_TIME(INT#12*TIME_TO_INT(tTmOut)), T#60s));
		TmOutTimer(IN := TRUE);

		(* send request *)
		fbRWData(
			NETID	:= aNetId,
			PORT	:= iProfinetPort,
			IDXGRP	:= iIGrp,
			IDXOFFS	:= 0,
			WRITELEN:= MIN(iDpv1ReqDataLen, iMAX_DPV1_SIZE_PNET_REQ),
			SRCADDR	:= pDpv1ReqData,
			READLEN	:= MIN(iDpv1ResDataLen, iMAX_DPV1_SIZE_PNET_RES),
			DESTADDR:= pDpv1ResData,
			WRTRD	:= FALSE,
			TMOUT	:= tTmOut
		);
		fbRWData(WRTRD	:= TRUE);

		iState := 1;
	END_IF

1:	(* write access data for DPV1 read request *)
	fbRWData(WRTRD	:= FALSE);

	IF NOT fbRWData.BUSY THEN
		fbRWData(WRTRD	:= FALSE);

		IF NOT fbRWData.ERR THEN
			(* read request parameter successfully sent, check for response *)
			WaitTimer(IN := FALSE);
			iState	:= 2; (* wait before polling *)
		ELSE
			bBusy	:= FALSE;
			bError	:= TRUE;
			iErrId	:= fbRWData.ERRID;
			IF ((UDINT_TO_DWORD(iErrId) AND DWORD#16#FF000000) = DWORD#16#27000000) THEN
				iErrorClass := UDINT_TO_BYTE(SHR((UDINT_TO_DWORD(iErrId) AND 16#00F00000), 20));
				iErrorCode := UDINT_TO_BYTE(SHR((UDINT_TO_DWORD(iErrId) AND 16#000F0000), 16));
			END_IF
			iState	:= 0;
		END_IF
	END_IF

2:	(* wait staate before next read response check *)
	WaitTimer(IN := TRUE, PT := tCommDelayDPV1PNET);
	IF WaitTimer.Q THEN
		stPNETFrameHeader.iRW := 0; (* read response *)

		(* read request parameter successfully sent, check for read response *)
		MEMSET(pDpv1ResData, 0, iMAX_DPV1_SIZE_PNET_RES);

		fbRWData(
			NETID	:= aNetId,
			PORT	:= iProfinetPort,
			IDXGRP	:= iIGrp,
			IDXOFFS	:= 0,
			WRITELEN:= SIZEOF(stPNETFrameHeader),
			SRCADDR	:= ADR(stPNETFrameHeader),
			READLEN	:= MIN(iDpv1ResDataLen, iMAX_DPV1_SIZE_PNET_RES),
			DESTADDR:= pDpv1ResData,
			WRTRD	:= FALSE,
			TMOUT	:= tTmOut
		);
		fbRWData(WRTRD	:= TRUE);
		iState	:= 3; (* CHECK READ *)
	END_IF

3:	(* wait for read response with data from DPV1 read request *)
	fbRWData(WRTRD := FALSE);

	IF NOT fbRWData.BUSY THEN
		fbRWData(WRTRD := FALSE);
		IF NOT fbRWData.ERR THEN
			MEMCPY(ADR(stDpv1ResHeader), pDpv1ResData, SIZEOF(stDpv1ResHeader));

			(* check for read response reference *)
			IF (stDpv1ResHeader.iRequestRef = stDpv1ReqHeader.iRequestRef) AND (stDpv1ResHeader.iAxis = stDpv1ReqHeader.iAxis) THEN
				(* response to last parameter request - split response data *)
				TmOutTimer(IN := FALSE);
				iState	:= 4; (* DONE *)
			ELSIF stDpv1ResHeader.iRequestRef = 0 THEN
				(* no response *)
				IF TmOutTimer.Q THEN
					(* complete read request timed out *)
					TmOutTimer(IN := FALSE);
					bBusy	:= FALSE;
					bError	:= TRUE;
					iErrId	:= 16#745; (* timeout *)
					iState	:= 0; (* ERROR *)
				ELSE
					(* no response, go to wait state *)
					WaitTimer(IN := FALSE);
					iState	:= 2; (* WAIT and REPEAT *)
				END_IF
			ELSE
				(* wrong response *)
				bBusy	:= FALSE;
				bError	:= TRUE;
				iErrId	:= 2; (* wrong reference response *)
				iState	:= 0; (* ERROR *)
			END_IF
		ELSE
			IF ((UDINT_TO_DWORD(fbRWData.ERRID) AND DWORD#16#FFFF0000) = DWORD#16#27B50000) OR ((UDINT_TO_DWORD(fbRWData.ERRID) AND DWORD#16#0000FFFF) = DWORD#16#00000723) THEN
				(* no response *)
				IF TmOutTimer.Q THEN
					(* complete read request timed out *)
					TmOutTimer(IN := FALSE);
					bBusy	:= FALSE;
					bError	:= TRUE;
					iErrId	:= 16#745; (* timeout *)
					iState	:= 0; (* ERROR *)
				ELSE
					(* no response, go to wait state *)
					WaitTimer(IN := FALSE);
					iState	:= 2; (* WAIT and REPEAT *)
				END_IF
			ELSE
				(* error *)
				bBusy	:= FALSE;
				bError	:= TRUE;
				iErrId	:= fbRWData.ERRID;
				IF ((UDINT_TO_DWORD(iErrId) AND DWORD#16#FF000000) = DWORD#16#27000000) THEN
					iErrorClass := UDINT_TO_BYTE(SHR((UDINT_TO_DWORD(iErrId) AND 16#00F00000), 20));
					iErrorCode := UDINT_TO_BYTE(SHR((UDINT_TO_DWORD(iErrId) AND 16#000F0000), 16));
				END_IF
				iState	:= 0; (* ERROR *)
			END_IF
		END_IF
	END_IF

4:	(* evaluate response *)
	IF stDpv1ResHeader.iRequestID = stDpv1ReqHeader.iRequestID THEN
		(* DPV1 Read successful - done *)
		bBusy	:= FALSE;
		iState	:= 0; (* DONE *)
	ELSIF (SINT_TO_BYTE(stDpv1ResHeader.iRequestID) AND 16#7F) = SINT_TO_BYTE(stDpv1ReqHeader.iRequestID) THEN
		(* DPV1 Read not successful or partly not successful *)
		bErrorValues:= TRUE;
		bBusy	:= FALSE;
		bError	:= TRUE;
		iErrId	:= 3; (* DPV1 Write not successful or partly not successful *)
		iState	:= 0; (* ERROR *)
	ELSE
		(* wrong response *)
		bBusy	:= FALSE;
		bError	:= TRUE;
		iErrId	:= 4; (* wrong response ID *)
		iState	:= 0; (* ERROR *)
	END_IF
END_CASE

(* clear flag *)
bExecute_ := bExecute_ AND bExecute;
END_FUNCTION_BLOCK

(* POU FB_GetDPRAMInfo, ST *)
FUNCTION_BLOCK FB_GetDPRAMInfo (*if the dpram must be accessed in a special manor, this function block returns error 0x701. In this case call FB_NovRamReadWriteEx to read data from the NOV-RAM and write data to the NOV-RAM.*)
VAR_INPUT
	nDevId 		: UDINT;		(* Device id of the FCxxxx or other DPRAM card ( Map the FC card as generic DPRAM/NOVRAM card im System Manager first ) *)
	bExecute		: BOOL;		(* Rising edge starts function block execution*)
	tTimeOut		: TIME := DEFAULT_ADS_TIMEOUT;	(* Max timeout for this command *)
END_VAR
VAR_OUTPUT
	bBusy 			: BOOL;
	bError			: BOOL;
	nErrid			: UDINT;
	stInfo			: ST_NovRamAddrInfo;
END_VAR
VAR
	FallingEdge		: F_TRIG;
	RisingRead		: R_TRIG;
	fbAdsReadEx	: ADSREADEX;
END_VAR
RisingRead( CLK := bExecute );
IF RisingRead.Q THEN
	bBusy := TRUE;
	bError := FALSE;
	nErrId := 0;
	MEMSET( ADR( stInfo ), 0, SIZEOF( stInfo ) );

	(* Get the nov ram address pointer and the novram byte size *)
	fbAdsReadEx( READ := FALSE );(*reset the fb*)
	fbAdsReadEx(
			NETID:= '',
			PORT:= AMSPORT_R0_IO,
			IDXGRP:= 16#5000+nDevId,
			IDXOFFS:= 16#FFFF_0200,
			LEN:= SIZEOF(stInfo),
			DESTADDR:= ADR(stInfo),
			READ:= TRUE,
			TMOUT:= tTimeout);
ELSE
		fbAdsReadEx( READ := FALSE );
END_IF

FallingEdge( CLK := fbAdsReadEx.BUSY );
IF FallingEdge.Q THEN
	bBusy := FALSE;
	IF NOT fbAdsReadEx.ERR THEN
		IF ( fbAdsReadEx.COUNT_R <> SIZEOF( stInfo ) ) THEN
			bError := TRUE;
			nErrId := 16#706;(* 1798 invalid parameter value(s)  *)
		END_IF
	ELSE
		bError := fbAdsReadEx.ERR;
		nErrId := fbAdsReadEx.ERRID;
	END_IF
END_IF
END_FUNCTION_BLOCK

(* POU FB_GetDPRAMInfoEx, ST *)
FUNCTION_BLOCK FB_GetDPRAMInfoEx
VAR_INPUT
	nDevId 		: UDINT;		(* Device id of the FCxxxx or other DPRAM card ( Map the FC card as generic DPRAM/NOVRAM card im System Manager first ) *)
	bExecute		: BOOL;		(* Rising edge starts function block execution*)
	tTimeOut		: TIME := DEFAULT_ADS_TIMEOUT;	(* Max timeout for this command *)
END_VAR
VAR_OUTPUT
	bBusy 			: BOOL;
	bError			: BOOL;
	nErrid			: UDINT;
	stInfo			: ST_NovRamAddrInfoEx;
END_VAR
VAR
	FallingEdge		: F_TRIG;
	RisingRead		: R_TRIG;
	fbAdsReadEx	: ADSREADEX;
END_VAR
RisingRead( CLK := bExecute );
IF RisingRead.Q THEN
	bBusy := TRUE;
	bError := FALSE;
	nErrId := 0;
	MEMSET( ADR( stInfo ), 0, SIZEOF( stInfo ) );

	(* Get the nov ram address pointer and the novram byte size *)

	(* Get the nov ram address pointer and the novram byte size *)
	fbAdsReadEx( READ := FALSE );(*reset the fb*)
	fbAdsReadEx(
		NETID:= '',
		PORT:= AMSPORT_R0_IO,
		IDXGRP:= 16#5000+nDevId,
		IDXOFFS:= 16#FFFF_0201,
		LEN:= MIN(SIZEOF( stInfo ), 10),
		DESTADDR:= ADR(stInfo),
		READ:= TRUE,
		TMOUT:= tTimeout);
ELSE
	fbAdsReadEx( READ := FALSE );
END_IF

FallingEdge( CLK := fbAdsReadEx.BUSY );
IF FallingEdge.Q THEN
	bBusy := FALSE;
	IF NOT fbAdsReadEx.ERR THEN
		IF ( fbAdsReadEx.COUNT_R <> MIN(SIZEOF( stInfo ), 10) ) THEN
			bError := TRUE;
			nErrId := 16#706;(* 1798 invalid parameter value(s)  *)
		END_IF
	ELSE
		bError := fbAdsReadEx.ERR;
		nErrId := fbAdsReadEx.ERRID;
	END_IF
END_IF
END_FUNCTION_BLOCK

(* POU FB_GetUPSStatus, ST *)
FUNCTION_BLOCK FB_GetUPSStatus
VAR_INPUT
	sNetId			: T_AmsNetId;
	nPort			: T_AmsPort := 0; (* 0 = Windows UPS service *)
	bEnable			: BOOL;
END_VAR
VAR_OUTPUT
	bValid			: BOOL;
	bError			: BOOL;
	nErrId			: UDINT;
	stStatus			:ST_UPSStatus;
END_VAR
{library private}
VAR
	fbRegQueryValue : FB_RegQueryValue;
	step				: INT;
	i				: INT;
	risingEdge		: R_TRIG;
	regNames		: ARRAY[1..11] OF STRING(25):=
(*  Config REG_SZ's *)					'Model', 'Vendor',
(*  Status REG_SZ's *)					'FirmwareRev', 'SerialNumber',
(*  Status REG_DWORD's *)				'CommStatus','BatteryCapacity','BatteryStatus','TotalUPSRuntime','TcPowerFailCnt', 'TcChargeFlags','UtilityPowerStatus';
	regSZData		: STRING;
	regDWData		: DWORD;

	delay			: TON := ( PT := T#300ms);
	tTimeOut			: TIME := T#2s;
	tmpStatus		:ST_UPSStatus;
	sPort	: STRING;
	sKey	: STRING;
END_VAR
risingEdge( CLK := bEnable );
IF risingEdge.Q THEN
	delay( IN := FALSE );
	bValid := FALSE;
	bError := FALSE;
	nErrId := 0;
(*	step := 1; *)
	step := -2;
	i := 0;
	MEMSET( ADR( stStatus ), 0, SIZEOF( stStatus) );
	fbRegQueryValue( bExecute := FALSE );
ELSIF NOT bEnable THEN
	step := 0;
END_IF

CASE step OF
	-2:
		fbRegQueryValue( bExecute := FALSE );
		fbRegQueryValue(sNetId:= sNetId, sSubKey:= 'Drivers\BuiltIn\Battery', sValName:='Port', cbData:=SIZEOF(sPort) , pData:=ADR(sPort) , bExecute:= TRUE , tTimeOut:=tTimeOut );
		step := -1;

	-1:
		fbRegQueryValue( bExecute := FALSE );
		IF NOT fbRegQueryValue.bBusy THEN
			IF NOT fbRegQueryValue.bError THEN
				sKey := 'Drivers\BuiltIn\Battery';
			ELSE
				sKey := 'SYSTEM\CurrentControlSet\Services\UPS';
			END_IF

			step := 1;
		END_IF



	0:	; (* idle step *)

	1:	(* Wait some time and repeat reading...*)
		delay( IN := TRUE );
		IF delay.Q THEN
			delay( IN := FALSE );
			i := i+1;
			step := step +1;
		END_IF
	2:
		fbRegQueryValue( bExecute := FALSE );
		CASE i OF
			1..2:
				fbRegQueryValue(sNetId:= sNetId, sSubKey:= CONCAT(sKey, '\Config'), sValName:=regNames[i], cbData:=SIZEOF(regSZData) , pData:=ADR(regSZData) , bExecute:= TRUE , tTimeOut:=tTimeOut );
			3..4:
				fbRegQueryValue(sNetId:= sNetId, sSubKey:= CONCAT(sKey, '\Status'), sValName:=regNames[i], cbData:=SIZEOF(regSZData) , pData:=ADR(regSZData) , bExecute:= TRUE , tTimeOut:=tTimeOut );
			5..11:
				fbRegQueryValue(sNetId:= sNetId, sSubKey:= CONCAT(sKey, '\Status'), sValName:=regNames[i], cbData:=SIZEOF(regDWData) , pData:=ADR(regDWData) , bExecute:= TRUE , tTimeOut:=tTimeOut );
		END_CASE
		step := step +1;
	3:
		fbRegQueryValue( bExecute := FALSE );
		IF NOT fbRegQueryValue.bBusy THEN
			IF NOT fbRegQueryValue.bError THEN
				CASE i OF
					1: tmpStatus.Model := regSZData;
					2: tmpStatus.Vendor := regSZData;
					3: tmpStatus.FirmwareRev := regSZData;
					4: tmpStatus.SerialNumber := regSZData;
					5: tmpStatus.eCommStatus := DWORD_TO_INT(regDWData);
					6: tmpStatus.BatteryLifePercent := regDWData;
					7: tmpStatus.eBatteryStatus := DWORD_TO_INT(regDWData);
					8: tmpStatus.BatteryLifeTime  := regDWData;
					9: tmpStatus.nPowerFailCnt  := regDWData;
					10: tmpStatus.dwChargeFlags :=  regDWData;
					11: tmpStatus.ePowerStatus := DWORD_TO_INT(regDWData);
						stStatus := tmpStatus;
						IF ( tmpStatus.Model =  ''  ) THEN
							bValid := FALSE;
							bError := TRUE;
							nErrId := 16#8001; (*UPS configuration error (no UPS configured?)*)
						ELSIF ( tmpStatus.eCommStatus <> UpsCommOk ) THEN
							bValid := FALSE;
							bError := TRUE;
							nErrId := 16#8002; (*UPS communication error (no communication to UPS?)*)
						ELSE
							bValid := TRUE;
							bError := FALSE;
							nErrId := 0; (* no error *)
						END_IF
						i := 0;
				END_CASE
			ELSE
				bValid := FALSE;
				bError := TRUE;
				IF ( ( fbRegQueryValue.nErrId = 1 ) OR ( fbRegQueryValue.nErrId = 2 ) ) THEN
					nErrId := 16#8003; (* Unknown error reading status data (status data not preset?)*)
				ELSE
					nErrId := fbRegQueryValue.nErrId;
				END_IF
				i := i - 1;
			END_IF
			step := 1;
		END_IF
END_CASE
END_FUNCTION_BLOCK

(* POU FB_KL1501Config, ST *)
FUNCTION_BLOCK FB_KL1501Config
VAR_INPUT
	bConfigurate			: BOOL; 		(*Rising edge starts configuration including read-configuration afterwards*)
	bReadConfig				: BOOL;			(*Rising edge reads the actual configuration*)
	iSetCounterType			: INT;			(*Counter-type to be set, see table*)
	bSetBackwardCounting	: BOOL;			(*Select backward-counting*)
	tTimeout				: TIME :=t#5s;	(*Time-out-time for Reading/Configuration - initially set to 5s*)
END_VAR
VAR_OUTPUT
	bBusy					: BOOL;			(*Reading or configuration is in progress*)
	bError					: BOOL;			(*Error while reading/configuration*)
	iErrorId				: UDINT;		(*Id of the last upcoming error*)
	iState					: USINT;		(*As long as the funcion-block is not busy, this variable shows the state of the terminal, otherwise it is 0*)
	iDataIn0				: UINT;			(*As long as the funcion-block is not busy, this variable shows the dataIn0 of the terminal, otherwise it keeps the value previous to reding/configuration*)
	iDataIn1				: UINT;			(*As long as the funcion-block is not busy, this variable shows the dataIn1 of the terminal, otherwise it keeps the value previous to reding/configuration*)
	iDataIn					: UDINT;		(*iDataIn1 and IDataIn0 put together as an UDINT, with iDataIn1 as High-Integer*)
	iTerminalType			: WORD;			(*Terminal-type-number, in this case 3228*)
	iSpecialType			: WORD;			(*Sub-type-number*)
	iFirmwareVersion		: WORD;			(*Firmware in ASCII-code*)
	sDescription			: STRING;		(*Terminal-type, special-type and firmware-version as readable text*)
	sCounterType			: STRING;		(*Text-description of entered counter-type*)
	bBackwardCounting		: BOOL;			(*TRUE: Backward-counting was selected*)
END_VAR
VAR
	rtRead					: R_TRIG;
	rtSet					: R_TRIG;
	bSetReq					: BOOL;
	tonTimeout				: TON;
	iStep					: INT;
	bSetConfigError			: BOOL;
	wReg32					: WORD;
	wSetReg32				: WORD;
	wFirmware				: WORD;
	pFirmware				: POINTER TO WORD;
	sFirmware				: STRING(2);
	iDataIn0Saved			: UINT;
	iDataIn1Saved			: UINT;
END_VAR
VAR_IN_OUT
	stInData   				: ST_KL1501InData;	(* Process image of the inputs. *)
	stOutData 				: ST_KL1501OutData;	(* Process image of the outputs. *)
END_VAR
tonTimeout	(PT:=tTimeout);
IF	tonTimeout.Q	THEN
	bError			:= TRUE;
	iErrorId		:= 16#8001;
	iStep			:= 0;
END_IF

rtSet	(CLK:=bConfigurate);
rtRead	(CLK:=bReadConfig);

IF	(rtSet.Q OR rtRead.Q)	AND NOT bBusy THEN
	bBusy			:= TRUE;
	bError			:= FALSE;
	iErrorId		:= 0;
	iDataIn0Saved	:= stInData.arrDataIn[0];
	iDataIn1Saved	:= stInData.arrDataIn[1];
	tonTimeout.IN	:= TRUE;
	iStep			:= 10;
	IF	rtSet.Q	THEN
		bSetReq	:= TRUE;
	END_IF
END_IF

IF bBusy THEN
	iDataIn0	:= iDataIn0Saved;
	iDataIn1	:= iDataIn1Saved;
	iState		:= 0;
ELSE
	iDataIn0	:= stInData.arrDataIn[0];
	iDataIn1	:= stInData.arrDataIn[1];
	iState		:= stInData.iState;
END_IF

iDataIn	:= UINT_TO_UDINT(iDataIn0)+(UINT_TO_UDINT(iDataIn1)*65536);

CASE iStep OF

0:	(*idle*)
	bBusy				:= FALSE;
	bSetReq				:= FALSE;
	tonTimeout.IN		:= FALSE;

10:	(*Klemmentyp (Kl32xx) auslesen: Register 8*)
	stOutData.iCtrl	:= 16#88;	(*Register 8 Lesen*)

	IF stInData.iState = 16#88 THEN
		iTerminalType	:= UINT_TO_WORD(stInData.arrDataIn[0]);
		iStep:=20;
	END_IF

20:	(*Spezialtyp (Kl1501-yyy) auslesen: Register 29*)
	stOutData.iCtrl	:= 16#9D;	(*Register 29 Lesen*)

	IF stInData.iState = 16#9D THEN
		iSpecialType	:= UINT_TO_WORD(stInData.arrDataIn[0]);
		iStep:=30;
	END_IF

30:	(*Firmware auslesen: Register 9*)
	stOutData.iCtrl	:= 16#89;	(*Register 9 Lesen*)

	IF stInData.iState = 16#89 THEN
		iFirmwareVersion:= UINT_TO_WORD(stInData.arrDataIn[0]);
		(*Umwandlung in STRING*)
		wFirmware		:= iFirmwareVersion;
		wFirmware		:= ROR(wFirmware,8);(*Reihenfolge der beiden Zeichen der Firmware tauschen*)
		pFirmware		:= ADR(sFirmware);	(*Einen Pointer auf den Info-String (Ausgang) legen*)
		pFirmware^		:= wFirmware;		(*Diesen Adressbereich mit dem richtig getauschen Wert beschreiben - damit ist auch der String beschrieben*)

		sDescription	:= CONCAT('Terminal ',WORD_TO_STRING(iTerminalType));

		CASE LEN(WORD_TO_STRING(iSpecialType)) OF
			1: sDescription	:= CONCAT(sDescription,'-000');
			2: sDescription	:= CONCAT(sDescription,'-00');
			3: sDescription	:= CONCAT(sDescription,'-0');
		ELSE
			sDescription	:= CONCAT(sDescription,'-');
		END_CASE

		sDescription	:= CONCAT(sDescription,WORD_TO_STRING(iSpecialType));
		sDescription	:= CONCAT(sDescription,' / Firmware ');
		sDescription	:= CONCAT(sDescription,sFirmware);

		IF bSetReq	THEN
			iStep:=100;
		ELSE
			iStep:=150;
		END_IF
	END_IF

	(*Falscher Klemmentyp angeschlossen, Konfiguration vorzeitig abbrechen*)
	IF (iTerminalType <> 1501)	THEN
		bError		:= TRUE;
		iErrorId	:= 16#8002;
		iStep		:= 160;
	END_IF
(*-----------------------------------------------------------------*)

100:(*jetzige Sensoreinstellung lesen: Register 32*)
	stOutData.iCtrl	:= 16#A0;	(*Register 32 Lesen*)

	IF stInData.iState = 16#A0 THEN
		wReg32			:= UINT_TO_WORD(stInData.arrDataIn[0]);
		A_SetConfigTable;			(*entsprechende Einstellungen vornehmen*)
		iStep:=110;
		IF	bSetConfigError	THEN
			iStep:=150;
		END_IF
	END_IF

110:(*Codewort Register 31 setzen: 16#1235 -> Schreibschutz aufheben*)
	stOutData.iCtrl	:= 16#DF;	(*Register 31 beschreiben*)
	stOutData.arrDataOut[0]	:= 16#1235;	(*Nutzdaten: Codewort*)

	IF stInData.iState = 16#9F THEN
		stOutData.iCtrl	:= 16#9F;	(*Register 31 Auslesen*)
		iStep:=120;
	END_IF

120:(*Bestätigung Codewort gesetzt erfragen*)
	IF	stInData.arrDataIn[0]	= 16#1235	THEN
		iStep:=130;
	END_IF

130:(*Nun Register 32 mit dem neuen Wert beschreiben*)
	stOutData.iCtrl	:= 16#E0;	(*Register 32 beschreiben*)
	stOutData.arrDataOut[0]	:= WORD_TO_UINT(wSetReg32);

	IF stInData.iState = 16#A0 THEN
		iStep:=140;
	END_IF

140:(*Codewort Register 31 löschen: 16#0000 -> Schreibschutz setzen*)
	stOutData.iCtrl	:= 16#DF;	(*Register 31 beschreiben*)
	stOutData.arrDataOut[0]	:= 16#0000;

	IF stInData.iState = 16#9F THEN
		iStep:=150;
	END_IF

150:(*nach erfolgter Parametrierung Sensoreinstellung lesen: Register 32*)
	stOutData.iCtrl	:= 16#A0;	(*Register 32 Lesen*)

	IF stInData.iState = 16#A0 THEN
		wReg32			:= UINT_TO_WORD(stInData.arrDataIn[0]);
		A_ReadConfigTable;
		iStep:=160;
	END_IF

160:(*Registerkommunikation beenden*)
	stOutData.iCtrl	:= 0; (*auch alle anderen Steuerbits mit ablöschen*)
	(*Rückmeldeabfrage Prozessdatenaustausch (Bit7) noch aktiv? *)
	(*alle anderen Bits könnten durch einen bestimmten Signalpegel gesetzt sein *)
	IF stInData.iState.7 = FALSE THEN
		iStep:=0;
	END_IF

END_CASE
END_FUNCTION_BLOCK
ACTION A_ReadConfigTable:
CASE (wReg32 AND 2#11100000000) OF	(*Check sensor-type via bits 8-10*)
	2#00100000000: sCounterType:='32-bit forward-backward-counter';
	2#01000000000: sCounterType:='Two 16-bit-forward-counter';
	2#10000000000: sCounterType:='32-bit gated forward-counter - Gate low inhibits';
	2#10100000000: sCounterType:='32-bit gated forward-counter - Gate high inhibits';
ELSE
	sCounterType:='Unknown';
	bError		:= TRUE;
	iErrorId	:= 16#8011;
END_CASE

bBackwardCounting:=wReg32.11;
END_ACTION
ACTION A_SetConfigTable:
bSetConfigError	:= FALSE;

wSetReg32:=wReg32 AND 2#1111000011111111;(*First clear the characteristical bits (8-11)*)

CASE iSetCounterType OF	(*Then set the counter-type via the bits 8-11*)

	0:	wSetReg32:=wSetReg32 OR 2#00100000000;(*32-bit forward-backward-counter*)
		wSetReg32.11:=bSetBackwardCounting;

	1:	wSetReg32:=wSetReg32 OR 2#01000000000;(*Two 16-bit-forward-counter*)
		wSetReg32.11:=bSetBackwardCounting;

	2:	wSetReg32:=wSetReg32 OR 2#10000000000;(*32-bit gated forward-counter - Gate low inhibits*)
		wSetReg32.11:=bSetBackwardCounting;

	3:	wSetReg32:=wSetReg32 OR 2#10100000000;(*32-bit gated forward-counter - Gate high inhibits*)
		wSetReg32.11:=bSetBackwardCounting;
ELSE
	bSetConfigError	:= TRUE;
	bError			:= TRUE;
	iErrorId		:= 16#8010;
END_CASE
END_ACTION

(* POU FB_KL27x1Config, ST *)
FUNCTION_BLOCK FB_KL27x1Config
VAR_INPUT
	bConfigurate			: BOOL; 		(*Rising edge starts configuration including read-configuration afterwards*)
	bReadConfig				: BOOL;			(*Rising edge reads the actual configuration*)
	bSetDimRampAbsolute		: BOOL;			(*FALSE: ramp-time refers to a step from 0..100%, TRUE: ramp-time refers to a step to the next value*)
	iSetRampTime			: INT;			(*Ramp-time to be set, see table*)
	bSetWatchdogDisable		: BOOL;			(*TRUE disables the watchdog for fieldbus-communication*)
	iSetWatchdogTimeout		: UINT;			(*Watchdog-time in 10ms-units*)
	iSetTimeoutOnValue		: UINT;			(*Value to be set, if timeout occurs and lamp was previously turned on*)
	iSetTimeoutOffValue		: UINT;			(*Value to be set, if timeout occurs and lamp was previously turned off*)
	iSetDimmerMode			: INT;			(*Dimmer-mode to be set, see table*)
	bSetOnAfterShortCircuit	: BOOL;			(*Selects, if the lamp has to be turned on after short-circuit*)
	bSetLineFrequency60Hz	: BOOL;			(*FALSE sets the line-frequency to 50Hz, TRUE to 60Hz*)
	tTimeout				: TIME :=t#5s;	(*Time-out-time for Reading/Configuration - initially set to 5s*)
END_VAR
VAR_OUTPUT
	bBusy					: BOOL;			(*Reading or configuration is in progress*)
	bError					: BOOL;			(*Error while reading/configuration*)
	iErrorId				: UDINT;		(*Id of the last upcoming error*)
	iState					: USINT;		(*As long as the funcion-block is not busy, this variable shows the state of the terminal, otherwise it is 0*)
	iTerminalType			: WORD;			(*Terminal-type-number, e.g. 2751*)
	iSpecialType			: WORD;			(*Sub-type-number*)
	iFirmwareVersion		: WORD;			(*Firmware in ASCII-code*)
	sDescription			: STRING;		(*Terminal-type, special-type and firmware-version as readable text*)

	bDimRampAbsolute		: BOOL;			(*TRUE: Dimramp was set to absolute - FALSE Dimramp was set to relative*)
	sRampTime				: STRING;		(*Ramp-time, which was set, according to the table*)
	bWatchdogDisable		: BOOL;			(*TRUE: Watchdog was disabled*)
	tWatchdogTimeout		: TIME;			(*Entered Watchdog-time*)
	iTimeoutOnValue			: UINT;			(*Timeout on-value, which was set*)
	iTimeoutOffValue		: UINT;			(*Timeout off-value, which was set*)
	sDimmerMode				: STRING;		(*Dimmer-mode, which was selected*)
	sAfterShortCircuit		: STRING;		(*Selected behaviour after short-circuit - on or off*)
	sLineFrequency			: STRING;		(*Selected line-frequency - 50 or 60 Hz*)
END_VAR
VAR
	rtRead					: R_TRIG;
	rtSet					: R_TRIG;
	bSetReq					: BOOL;
	tonTimeout				: TON;
	iStep					: INT;
	bSetConfigError			: BOOL;
	wReg32					: WORD;
	wSetReg32				: WORD;
	wReg35					: WORD;
	wSetReg35				: WORD;
	wReg36					: WORD;
	wSetReg36				: WORD;
	wReg37					: WORD;
	wSetReg37				: WORD;
	wReg38					: WORD;
	wSetReg38				: WORD;
	wReg39					: WORD;
	wSetReg39				: WORD;
	wReg40					: WORD;
	wSetReg40				: WORD;
	wReg41					: WORD;
	wSetReg41				: WORD;
	wFirmware				: WORD;
	pFirmware				: POINTER TO WORD;
	sFirmware				: STRING(2);
END_VAR
VAR_IN_OUT
	stInData   				: ST_KL27x1InData;	(* Process image of the inputs. *)
	stOutData 				: ST_KL27x1OutData;	(* Process image of the outputs. *)
END_VAR
tonTimeout	(PT:=tTimeout);
IF	tonTimeout.Q	THEN
	bError			:= TRUE;
	iErrorId		:= 16#8001;
	iStep			:= 0;
END_IF

rtSet	(CLK:=bConfigurate);
rtRead	(CLK:=bReadConfig);

IF	(rtSet.Q OR rtRead.Q)	AND NOT bBusy THEN
	bBusy			:= TRUE;
	bError			:= FALSE;
	iErrorId		:= 0;
	tonTimeout.IN	:= TRUE;
	iStep			:= 10;
	IF	rtSet.Q	THEN
		bSetReq	:= TRUE;
	END_IF
END_IF

IF bBusy THEN
	iState		:= 0;
ELSE
	iState		:= stInData.iState;
END_IF


CASE iStep OF

0:	(*idlde*)
	bBusy				:= FALSE;
	bSetReq				:= FALSE;
	tonTimeout.IN		:= FALSE;

10:	(*Klemmentyp (Kl27xx) auslesen: Register 8*)
	stOutData.iCtrl	:= 16#88;	(*Register 8 Lesen*)

	IF stInData.iState = 16#88 THEN
		iTerminalType	:= INT_TO_WORD(stInData.iDataIn);
		iStep:=20;
	END_IF

20:	(*Spezialtyp (Kl27xx-yyy) auslesen: Register 29*)
	stOutData.iCtrl	:= 16#9D;	(*Register 29 Lesen*)

	IF stInData.iState = 16#9D THEN
		iSpecialType	:= INT_TO_WORD(stInData.iDataIn);
		iStep:=30;
	END_IF

30:	(*Firmware auslesen: Register 9*)
	stOutData.iCtrl	:= 16#89;	(*Register 9 Lesen*)

	IF stInData.iState = 16#89 THEN
		iFirmwareVersion:= INT_TO_WORD(stInData.iDataIn);
		(*Umwandlung in STRING*)
		wFirmware		:= iFirmwareVersion;
		wFirmware		:= ROR(wFirmware,8);(*Reihenfolge der beiden Zeichen der Firmware tauschen*)
		pFirmware		:= ADR(sFirmware);	(*Einen Pointer auf den Info-String (Ausgang) legen*)
		pFirmware^		:= wFirmware;		(*Diesen Adressbereich mit dem richtig getauschen Wert beschreiben - damit ist auch der String beschrieben*)

		sDescription	:= CONCAT('Terminal ',WORD_TO_STRING(iTerminalType));

		CASE LEN(WORD_TO_STRING(iSpecialType)) OF
			1: sDescription	:= CONCAT(sDescription,'-000');
			2: sDescription	:= CONCAT(sDescription,'-00');
			3: sDescription	:= CONCAT(sDescription,'-0');
		ELSE
			sDescription	:= CONCAT(sDescription,'-');
		END_CASE

		sDescription	:= CONCAT(sDescription,WORD_TO_STRING(iSpecialType));
		sDescription	:= CONCAT(sDescription,' / Firmware ');
		sDescription	:= CONCAT(sDescription,sFirmware);

		IF bSetReq	THEN
			iStep:=100;
		ELSE
			iStep:=150;
		END_IF
	END_IF

	(*Falscher Klemmentyp angeschlossen, Konfiguration vorzeitig abbrechen*)
	IF ((iTerminalType <> 2751)	AND (iTerminalType <> 2761))	THEN
		bError		:= TRUE;
		iErrorId	:= 16#8002;
		iStep		:= 160;
	END_IF

(*-----------------------------------------------------------------*)

100:(*jetzige Sensoreinstellung lesen: Register 32*)
	stOutData.iCtrl	:= 16#A0;	(*Register 32 Lesen*)

	IF stInData.iState = 16#A0 THEN
		wReg32			:= INT_TO_WORD(stInData.iDataIn);
		A_SetConfigTable;			(*entsprechende Einstellungen vornehmen*)
		iStep:=110;
		IF	bSetConfigError	THEN
			iStep:=150;
		END_IF
	END_IF

110:(*Codewort Register 31 setzen: 16#1235 -> Schreibschutz aufheben*)
	stOutData.iCtrl	:= 16#DF;	(*Register 31 beschreiben*)
	stOutData.iDataOut	:= 16#1235;	(*Nutzdaten: Codewort*)

	IF stInData.iState = 16#9F THEN
		stOutData.iCtrl	:= 16#9F;	(*Register 31 Auslesen*)
		iStep:=120;
	END_IF

120:(*Bestätigung Codewort gesetzt erfragen*)
	IF	stInData.iDataIn	= 16#1235	THEN
		iStep:=130;
	END_IF

130:(*Register 32 mit dem neuen Wert beschreiben*)
	stOutData.iCtrl	:= 16#E0;	(*Register 32 beschreiben*)
	stOutData.iDataOut	:= WORD_TO_INT(wSetReg32);

	IF stInData.iState = 16#A0 THEN
		iStep:=131;
	END_IF

131:(*Register 35 mit dem neuen Wert beschreiben*)
	stOutData.iCtrl	:= 16#E3;	(*Register 35 beschreiben*)
	stOutData.iDataOut	:= WORD_TO_INT(wSetReg35);

	IF stInData.iState = 16#A3 THEN
		iStep:=132;
	END_IF

132:(*Register 36 mit dem neuen Wert beschreiben*)
	stOutData.iCtrl	:= 16#E4;	(*Register 36 beschreiben*)
	stOutData.iDataOut	:= WORD_TO_INT(wSetReg36);

	IF stInData.iState = 16#A4 THEN
		iStep:=133;
	END_IF

133:(*Register 37 mit dem neuen Wert beschreiben*)
	stOutData.iCtrl	:= 16#E5;	(*Register 37 beschreiben*)
	stOutData.iDataOut	:= WORD_TO_INT(wSetReg37);

	IF stInData.iState = 16#A5 THEN
		iStep:=134;
	END_IF

134:(*Register 38 mit dem neuen Wert beschreiben*)
	stOutData.iCtrl	:= 16#E6;	(*Register 38 beschreiben*)
	stOutData.iDataOut	:= WORD_TO_INT(wSetReg38);

	IF stInData.iState = 16#A6 THEN
		iStep:=135;
	END_IF

135:(*Register 39 mit dem neuen Wert beschreiben*)
	stOutData.iCtrl	:= 16#E7;	(*Register 39 beschreiben*)
	stOutData.iDataOut	:= WORD_TO_INT(wSetReg39);

	IF stInData.iState = 16#A7 THEN
		iStep:=136;
	END_IF

136:(*Register 40 mit dem neuen Wert beschreiben*)
	stOutData.iCtrl	:= 16#E8;	(*Register 40 beschreiben*)
	stOutData.iDataOut	:= WORD_TO_INT(wSetReg40);

	IF stInData.iState = 16#A8 THEN
		iStep:=137;
	END_IF

137:(*Register 41 mit dem neuen Wert beschreiben*)
	stOutData.iCtrl	:= 16#E9;	(*Register 41 beschreiben*)
	stOutData.iDataOut	:= WORD_TO_INT(wSetReg41);

	IF stInData.iState = 16#A9 THEN
		iStep:=140;
	END_IF

140:(*Codewort Register 31 löschen: 16#0000 -> Schreibschutz setzen*)
	stOutData.iCtrl	:= 16#DF;	(*Register 31 beschreiben*)
	stOutData.iDataOut	:= 16#0000;

	IF stInData.iState = 16#9F THEN
		iStep:=150;
	END_IF

150:(*nach erfolgter Parametrierung Konfiguration lesen: Register 32*)
	stOutData.iCtrl	:= 16#A0;	(*Register 32 Lesen*)

	IF stInData.iState = 16#A0 THEN
		wReg32			:= INT_TO_WORD(stInData.iDataIn);
		iStep:=151;
	END_IF

151:(*nach erfolgter Parametrierung Konfiguration lesen: Register 35*)
	stOutData.iCtrl	:= 16#A3;	(*Register 35 Lesen*)

	IF stInData.iState = 16#A3 THEN
		wReg35			:= INT_TO_WORD(stInData.iDataIn);
		iStep:=152;
	END_IF

152:(*nach erfolgter Parametrierung Konfiguration lesen: Register 36*)
	stOutData.iCtrl	:= 16#A4;	(*Register 36 Lesen*)

	IF stInData.iState = 16#A4 THEN
		wReg36			:= INT_TO_WORD(stInData.iDataIn);
		iStep:=153;
	END_IF

153:(*nach erfolgter Parametrierung Konfiguration lesen: Register 37*)
	stOutData.iCtrl	:= 16#A5;	(*Register 37 Lesen*)

	IF stInData.iState = 16#A5 THEN
		wReg37			:= INT_TO_WORD(stInData.iDataIn);
		iStep:=154;
	END_IF

154:(*nach erfolgter Parametrierung Konfiguration lesen: Register 38*)
	stOutData.iCtrl	:= 16#A6;	(*Register 38 Lesen*)

	IF stInData.iState = 16#A6 THEN
		wReg38			:= INT_TO_WORD(stInData.iDataIn);
		iStep:=155;
	END_IF

155:(*nach erfolgter Parametrierung Konfiguration lesen: Register 39*)
	stOutData.iCtrl	:= 16#A7;	(*Register 39 Lesen*)

	IF stInData.iState = 16#A7 THEN
		wReg39			:= INT_TO_WORD(stInData.iDataIn);
		iStep:=156;
	END_IF

156:(*nach erfolgter Parametrierung Konfiguration lesen: Register 40*)
	stOutData.iCtrl	:= 16#A8;	(*Register 40 Lesen*)

	IF stInData.iState = 16#A8 THEN
		wReg40			:= INT_TO_WORD(stInData.iDataIn);
		iStep:=157;
	END_IF


157:(*nach erfolgter Parametrierung Konfiguration lesen: Register 41*)
	stOutData.iCtrl	:= 16#A9;	(*Register 41 Lesen*)

	IF stInData.iState = 16#A9 THEN
		wReg41			:= INT_TO_WORD(stInData.iDataIn);
		A_ReadConfigTable;
		iStep:=160;
	END_IF


160:(*Registerkommunikation beenden*)
	stOutData.iCtrl	:= 0; (*auch alle anderen Steuerbits mit ablöschen*)
	(*Rückmeldeabfrage Prozessdatenaustausch (Bit7) noch aktiv? *)
	(*alle anderen Bits könnten durch einen bestimmten Signalpegel gesetzt sein *)
	IF stInData.iState.7 = FALSE THEN
		iStep:=0;
	END_IF

END_CASE
END_FUNCTION_BLOCK
ACTION A_ReadConfigTable:
bWatchdogDisable	:= wReg32.2;
bDimRampAbsolute	:= wReg32.3;


CASE wReg35 OF
	0:	sRampTime	:= '50 ms';
	1:	sRampTime	:= '100 ms';
	2:	sRampTime	:= '200 ms';
	3:	sRampTime	:= '500 ms';
	4:	sRampTime	:= '1 s';
	5:	sRampTime	:= '2 s';
	6:	sRampTime	:= '5 s';
	7:	sRampTime	:= '10 s';
ELSE
	sRampTime	:= 'unknown register-entry';
	bError		:= TRUE;
	iErrorId	:= 16#801A;
END_CASE


tWatchdogTimeout	:= WORD_TO_TIME(wReg36)*10;
iTimeoutOnValue		:= wReg37;
iTimeoutOffValue	:= wReg38;


CASE wReg39 OF
	0:	sDimmerMode	:= '0 - Automatic recognition';
	1:	sDimmerMode	:= '1 - Trailing phase angle';
	2:	sDimmerMode	:= '2 - Leading phase angle';
	3:	sDimmerMode	:= '3 - Rectifier mode, positive';
	4:	sDimmerMode	:= '4 - Rectifier mode, negative';
ELSE
	sDimmerMode	:= 'unknown register-entry';
	bError		:= TRUE;
	iErrorId	:= 16#801B;
END_CASE


CASE wReg40 OF
	0:	sAfterShortCircuit := 'Off';
	1:	sAfterShortCircuit := 'On';
ELSE
	sAfterShortCircuit	:= 'unknown register-entry';
	bError				:= TRUE;
	iErrorId			:= 16#801C;
END_CASE


CASE wReg41 OF
	0:	sLineFrequency := '50 Hz';
	1:	sLineFrequency := '60 Hz';
ELSE
	sLineFrequency	:= 'unknown register-entry';
	bError			:= TRUE;
	iErrorId		:= 16#801D;
END_CASE
END_ACTION
ACTION A_SetConfigTable:
bSetConfigError	:= FALSE;

wSetReg32	:= wReg32	AND 2#1111111111110011;(*Clear bits 2 and 3 of Reg32*)
wSetReg32.2	:= bSetWatchdogDisable;
wSetReg32.3	:= bSetDimRampAbsolute;

CASE iSetRampTime OF
	0:	wSetReg35	:= 0;		(*50 ms*)
	1:	wSetReg35	:= 1;		(*100 ms*)
	2:	wSetReg35	:= 2;		(*200 ms*)
	3:	wSetReg35	:= 3;		(*500 ms*)
	4:	wSetReg35	:= 4;		(*1 s*)
	5:	wSetReg35	:= 5;		(*2 s*)
	6:	wSetReg35	:= 6;		(*5 s*)
	7:	wSetReg35	:= 7;		(*10 s*)
ELSE
	bSetConfigError	:= TRUE;
	bError			:= TRUE;
	iErrorId		:= 16#8018;
END_CASE


wSetReg36	:=	UINT_TO_WORD(iSetWatchdogTimeout);
wSetReg37	:=	UINT_TO_WORD(iSetTimeoutOnValue);
wSetReg38	:=	UINT_TO_WORD(iSetTimeoutOffValue);


CASE iSetDimmerMode OF
	0:	wSetReg39	:= 0;		(*automatic recognition*)
	1:	wSetReg39	:= 1;		(*trailing phase angle*)
	2:	wSetReg39	:= 2;		(*leading phase angle*)
	3:	wSetReg39	:= 3;		(*Rectifier mode, positive*)
	4:	wSetReg39	:= 4;		(*Rectifier mode, negative*)
ELSE
	bSetConfigError	:= TRUE;
	bError			:= TRUE;
	iErrorId		:= 16#8019;
END_CASE

IF	bSetOnAfterShortCircuit	THEN
		wSetReg40	:= 1;
ELSE	wSetReg40	:= 0;
END_IF

IF	bSetLineFrequency60Hz	THEN
		wSetReg41	:= 1;
ELSE	wSetReg41	:= 0;
END_IF
END_ACTION

